KUKA KRL program: EPS_2_25089_SANMH01A_C_20251118074754.src

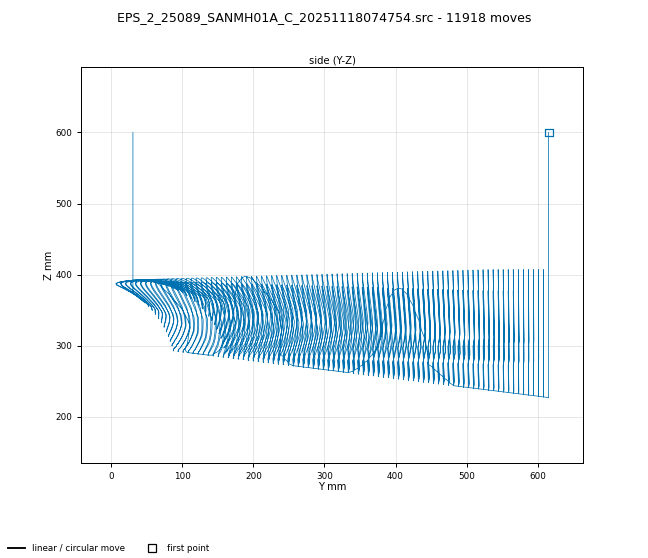
[picture p0: tool path of EPS_2_25089_SANMH01A_C_20251118074754.src, 11918 of 11920 moves have a stored position in this frame; points joined in program order, loops and branches not executed]
&ACCESS RVP
&REL 4
&COMMENT QRS 19112012
&PARAM EDITMASK = *
DEF PART()
EXT BAS (BAS_COMMAND :IN,REAL :IN )
INT I
BAS (#INITMOV,0 )

;KUKA QRS Post kuka4.cps  Date:22-06-2017 !

File_ID=2924

QRS_PRE_INIT()

;Init var - Until changes are made in qrs_pre_init
Outlet_Square_prg=0
Inlet_1_Square_prg=0
Inlet_2_Square_prg=0
Inlet_3_Square_prg=0
Inlet_4_Square_prg=0
Inlet_5_Square_prg=0

Outlet_1={X 0.000, Y 531.880, Z 306.500, B 0.000, E1 0.000 }
Inlet_1={X 0.000, Y 534.050, Z 276.500, B 0.000, E1 193.000 }
Outlet_1_type=201
Inlet_1_type=201
;QRS#1=Sidecore dimensions
;QRS#2=200-8" PVC SDR 35
;QRS#3=200-8" PVC SDR 35
;QRS#4=
;QRS#5=
;QRS#6=
;QRS#7=
;QRS#8=
;QRS#9=12-08 PSX
;QRS#10=12-08 PSX
;QRS#11=
;QRS#12=
;QRS#13=
;QRS#14=
;QRS#15=
;QRS#16=1220x127x686 2,25'
;QRS#17=EPS Height
;QRS#18=407
;QRS#19=*
;QRS#20= UPDATED VERSION 22-06-2017
;QRS#21=*
Outlet_Square=0100
Inlet_1_Square=0100
Inlet_2_Square=0
Inlet_3_Square=0
Inlet_4_Square=0
Inlet_5_Square=0
Mill_Square=1
Outlet_Square_Prg=204
Inlet_1_Square_prg=204

QRS_INIT()

$ADVANCE=5

; T1
PTP {E1 173.593,E2 173.593}
PTP {X 0,Y 615.507,A -85,B 0,C 180,E1 173.593,E2 173.593,E3 0,E4 0,E5 0,E6 0}
QRS_SPEED_INIT()
LIN {X 0,Y 615.507,Z 600,A -85,B 0,C 180,E1 173.593,E2 173.593,E3 0,E4 0,E5 0,E6 0} C_VEL
LIN {X 0,Y 615.507,Z 236.874,A -85,B 0,C 180,E1 173.593,E2 173.593} C_VEL
LIN {X 0,Y 615.507,Z 228.699,A -85,B 0,C 180,E1 173.593,E2 173.593} C_VEL
LIN {X 0,Y 615.492,Z 226.699,A -85,B 0,C 180,E1 173.407,E2 173.407} C_VEL
LIN {X 0,Y 615.497,Z 226.682,A -85,B 0,C 180,E1 170.802,E2 170.802} C_VEL
LIN {X 0,Y 615.47,Z 226.694,A -85,B 0,C 180,E1 168.14,E2 168.14} C_VEL
LIN {X 0,Y 615.478,Z 226.693,A -85,B 0,C 180,E1 165.452,E2 165.452} C_VEL
LIN {X 0,Y 615.483,Z 226.686,A -85,B 0,C 180,E1 162.73,E2 162.73} C_VEL
LIN {X 0,Y 615.486,Z 226.7,A -85,B 0,C 180,E1 159.968,E2 159.968} C_VEL
LIN {X 0,Y 615.487,Z 226.684,A -85,B 0,C 180,E1 157.157,E2 157.157} C_VEL
LIN {X 0,Y 615.497,Z 226.7,A -85,B 0,C 180,E1 154.286,E2 154.286} C_VEL
LIN {X 0,Y 615.486,Z 226.684,A -85,B 0,C 180,E1 151.343,E2 151.343} C_VEL
LIN {X 0,Y 615.486,Z 226.692,A -85,B 0,C 180,E1 148.912,E2 148.912} C_VEL
LIN {X 0,Y 615.482,Z 226.698,A -85,B 0,C 180,E1 146.465,E2 146.465} C_VEL
LIN {X 0,Y 615.482,Z 226.685,A -85,B 0,C 180,E1 143.576,E2 143.576} C_VEL
LIN {X 0,Y 615.497,Z 226.699,A -85,B 0,C 180,E1 140.935,E2 140.935} C_VEL
LIN {X 0,Y 615.464,Z 226.694,A -85,B 0,C 180,E1 138.526,E2 138.526} C_VEL
LIN {X 0,Y 615.487,Z 226.685,A -85,B 0,C 180,E1 135.852,E2 135.852} C_VEL
LIN {X 0,Y 615.478,Z 226.699,A -85,B 0,C 180,E1 133.048,E2 133.048} C_VEL
LIN {X 0,Y 615.453,Z 226.693,A -85,B 0,C 180,E1 130.608,E2 130.608} C_VEL
LIN {X 0,Y 615.48,Z 226.689,A -85,B 0,C 180,E1 128.013,E2 128.013} C_VEL
LIN {X 0,Y 615.496,Z 226.699,A -85,B 0,C 180,E1 125.614,E2 125.614} C_VEL
LIN {X 0,Y 615.458,Z 226.697,A -85,B 0,C 180,E1 123.237,E2 123.237} C_VEL
LIN {X 0,Y 615.443,Z 226.694,A -85,B 0,C 180,E1 120.921,E2 120.921} C_VEL
LIN {X 0,Y 615.471,Z 226.691,A -85,B 0,C 180,E1 118.45,E2 118.45} C_VEL
LIN {X 0,Y 615.454,Z 226.698,A -85,B 0,C 180,E1 115.565,E2 115.565} C_VEL
LIN {X 0,Y 615.445,Z 226.698,A -85,B 0,C 180,E1 113.558,E2 113.558} C_VEL
LIN {X 0,Y 615.493,Z 226.694,A -85,B 0,C 180,E1 112.351,E2 112.351} C_VEL
LIN {X 0,Y 615.457,Z 230.7,A -85,B 0,C 180,E1 110.033,E2 110.033} C_VEL
LIN {X 0,Y 615.474,Z 234.384,A -85,B 0,C 180,E1 107.957,E2 107.957} C_VEL
LIN {X 0,Y 615.463,Z 239.321,A -85,B 0,C 180,E1 105.226,E2 105.226} C_VEL
LIN {X 0,Y 615.494,Z 244.376,A -85,B 0,C 180,E1 102.53,E2 102.53} C_VEL
LIN {X 0,Y 615.48,Z 249.482,A -85,B 0,C 180,E1 99.862,E2 99.862} C_VEL
LIN {X 0,Y 615.464,Z 254.653,A -85,B 0,C 180,E1 97.216,E2 97.216} C_VEL
LIN {X 0,Y 615.491,Z 259.883,A -85,B 0,C 180,E1 94.584,E2 94.584} C_VEL
LIN {X 0,Y 615.468,Z 265.156,A -85,B 0,C 180,E1 91.963,E2 91.963} C_VEL
LIN {X 0,Y 615.47,Z 270.494,A -85,B 0,C 180,E1 89.346,E2 89.346} C_VEL
LIN {X 0,Y 615.49,Z 272.087,A -85,B 0,C 180,E1 88.569,E2 88.569} C_VEL
LIN {X 0,Y 615.475,Z 287.993,A -85,B 0,C 180,E1 88.201,E2 88.201} C_VEL
LIN {X 0,Y 615.457,Z 299.97,A -85,B 0,C 180,E1 87.791,E2 87.791} C_VEL
LIN {X 0,Y 615.485,Z 312.305,A -85,B 0,C 180,E1 87.218,E2 87.218} C_VEL
LIN {X 0,Y 615.497,Z 323.338,A -85,B 0,C 180,E1 86.563,E2 86.563} C_VEL
LIN {X 0,Y 615.498,Z 333.348,A -85,B 0,C 180,E1 85.826,E2 85.826} C_VEL
LIN {X 0,Y 615.497,Z 343.183,A -85,B 0,C 180,E1 84.923,E2 84.923} C_VEL
LIN {X 0,Y 615.497,Z 351.875,A -85,B 0,C 180,E1 83.937,E2 83.937} C_VEL
LIN {X 0,Y 615.498,Z 357.916,A -85,B 0,C 180,E1 83.094,E2 83.094} C_VEL
LIN {X 0,Y 615.495,Z 363.597,A -85,B 0,C 180,E1 82.125,E2 82.125} C_VEL
LIN {X 0,Y 615.498,Z 368.188,A -85,B 0,C 180,E1 81.133,E2 81.133} C_VEL
LIN {X 0,Y 615.496,Z 371.686,A -85,B 0,C 180,E1 80.138,E2 80.138} C_VEL
LIN {X 0,Y 615.496,Z 374.268,A -85,B 0,C 180,E1 79.101,E2 79.101} C_VEL
LIN {X 0,Y 615.494,Z 375.727,A -85,B 0,C 180,E1 78.14,E2 78.14} C_VEL
LIN {X 0,Y 615.497,Z 376.266,A -85,B 0,C 180,E1 77.47,E2 77.47} C_VEL
LIN {X 0,Y 615.495,Z 376.357,A -85,B 0,C 180,E1 76.799,E2 76.799} C_VEL
LIN {X 0,Y 615.497,Z 376.002,A -85,B 0,C 180,E1 76.058,E2 76.058} C_VEL
LIN {X 0,Y 615.496,Z 375.351,A -85,B 0,C 180,E1 75.452,E2 75.452} C_VEL
LIN {X 0,Y 615.495,Z 374.193,A -85,B 0,C 180,E1 74.775,E2 74.775} C_VEL
LIN {X 0,Y 615.494,Z 371.016,A -85,B 0,C 180,E1 73.562,E2 73.562} C_VEL
LIN {X 0,Y 615.498,Z 366.514,A -85,B 0,C 180,E1 72.387,E2 72.387} C_VEL
LIN {X 0,Y 615.497,Z 361.234,A -85,B 0,C 180,E1 71.355,E2 71.355} C_VEL
LIN {X 0,Y 615.496,Z 354.453,A -85,B 0,C 180,E1 70.316,E2 70.316} C_VEL
LIN {X 0,Y 615.494,Z 345.883,A -85,B 0,C 180,E1 69.27,E2 69.27} C_VEL
LIN {X 0,Y 615.497,Z 336.964,A -85,B 0,C 180,E1 68.393,E2 68.393} C_VEL
LIN {X 0,Y 615.499,Z 325.956,A -85,B 0,C 180,E1 67.526,E2 67.526} C_VEL
LIN {X 0,Y 615.442,Z 315.935,A -85,B 0,C 180,E1 66.888,E2 66.888} C_VEL
LIN {X 0,Y 615.437,Z 303.663,A -85,B 0,C 180,E1 66.274,E2 66.274} C_VEL
LIN {X 0,Y 615.477,Z 290.8,A -85,B 0,C 180,E1 65.795,E2 65.795} C_VEL
LIN {X 0,Y 615.485,Z 277.91,A -85,B 0,C 180,E1 65.459,E2 65.459} C_VEL
LIN {X 0,Y 615.477,Z 272.101,A -85,B 0,C 180,E1 65.346,E2 65.346} C_VEL
LIN {X 0,Y 615.431,Z 266.947,A -85,B 0,C 180,E1 62.821,E2 62.821} C_VEL
LIN {X 0,Y 615.43,Z 262.428,A -85,B 0,C 180,E1 60.591,E2 60.591} C_VEL
LIN {X 0,Y 615.447,Z 257.861,A -85,B 0,C 180,E1 58.313,E2 58.313} C_VEL
LIN {X 0,Y 615.494,Z 253.242,A -85,B 0,C 180,E1 55.979,E2 55.979} C_VEL
LIN {X 0,Y 615.46,Z 248.58,A -85,B 0,C 180,E1 53.574,E2 53.574} C_VEL
LIN {X 0,Y 615.424,Z 243.841,A -85,B 0,C 180,E1 51.092,E2 51.092} C_VEL
LIN {X 0,Y 615.425,Z 239.751,A -85,B 0,C 180,E1 48.91,E2 48.91} C_VEL
LIN {X 0,Y 615.468,Z 235.816,A -85,B 0,C 180,E1 46.755,E2 46.755} C_VEL
LIN {X 0,Y 615.484,Z 230.919,A -85,B 0,C 180,E1 43.998,E2 43.998} C_VEL
LIN {X 0,Y 615.492,Z 227.552,A -85,B 0,C 180,E1 42.082,E2 42.082} C_VEL
LIN {X 0,Y 615.47,Z 226.699,A -85,B 0,C 180,E1 41.474,E2 41.474} C_VEL
LIN {X 0,Y 615.479,Z 226.701,A -85,B 0,C 180,E1 38.904,E2 38.904} C_VEL
LIN {X 0,Y 615.487,Z 226.691,A -85,B 0,C 180,E1 36.423,E2 36.423} C_VEL
LIN {X 0,Y 615.475,Z 226.7,A -85,B 0,C 180,E1 34.021,E2 34.021} C_VEL
LIN {X 0,Y 615.495,Z 226.698,A -85,B 0,C 180,E1 31.089,E2 31.089} C_VEL
LIN {X 0,Y 615.49,Z 226.695,A -85,B 0,C 180,E1 28.453,E2 28.453} C_VEL
LIN {X 0,Y 615.459,Z 226.7,A -85,B 0,C 180,E1 25.566,E2 25.566} C_VEL
LIN {X 0,Y 615.49,Z 226.69,A -85,B 0,C 180,E1 22.843,E2 22.843} C_VEL
LIN {X 0,Y 615.449,Z 226.7,A -85,B 0,C 180,E1 20.033,E2 20.033} C_VEL
LIN {X 0,Y 615.488,Z 226.694,A -85,B 0,C 180,E1 17.269,E2 17.269} C_VEL
LIN {X 0,Y 615.485,Z 226.702,A -85,B 0,C 180,E1 14.548,E2 14.548} C_VEL
LIN {X 0,Y 615.469,Z 226.7,A -85,B 0,C 180,E1 11.86,E2 11.86} C_VEL
LIN {X 0,Y 615.497,Z 226.689,A -85,B 0,C 180,E1 9.198,E2 9.198} C_VEL
LIN {X 0,Y 615.453,Z 226.7,A -85,B 0,C 180,E1 6.556,E2 6.556} C_VEL
LIN {X 0,Y 615.49,Z 226.699,A -85,B 0,C 180,E1 3.928,E2 3.928} C_VEL
LIN {X 0,Y 615.496,Z 226.694,A -85,B 0,C 180,E1 1.308,E2 1.308} C_VEL
LIN {X 0,Y 615.447,Z 226.7,A -85,B 0,C 180,E1 -1.309,E2 -1.309} C_VEL
LIN {X 0,Y 615.479,Z 226.695,A -85,B 0,C 180,E1 -3.929,E2 -3.929} C_VEL
LIN {X 0,Y 615.487,Z 226.701,A -85,B 0,C 180,E1 -6.589,E2 -6.589} C_VEL
LIN {X 0,Y 615.47,Z 226.698,A -85,B 0,C 180,E1 -9.2,E2 -9.2} C_VEL
LIN {X 0,Y 615.478,Z 226.693,A -85,B 0,C 180,E1 -11.862,E2 -11.862} C_VEL
LIN {X 0,Y 615.458,Z 226.699,A -85,B 0,C 180,E1 -14.55,E2 -14.55} C_VEL
LIN {X 0,Y 615.487,Z 226.698,A -85,B 0,C 180,E1 -17.271,E2 -17.271} C_VEL
LIN {X 0,Y 615.493,Z 226.699,A -85,B 0,C 180,E1 -20.033,E2 -20.033} C_VEL
LIN {X 0,Y 615.475,Z 226.698,A -85,B 0,C 180,E1 -22.846,E2 -22.846} C_VEL
LIN {X 0,Y 615.493,Z 226.692,A -85,B 0,C 180,E1 -25.716,E2 -25.716} C_VEL
LIN {X 0,Y 615.456,Z 226.699,A -85,B 0,C 180,E1 -28.66,E2 -28.66} C_VEL
LIN {X 0,Y 615.48,Z 226.695,A -85,B 0,C 180,E1 -31.087,E2 -31.087} C_VEL
LIN {X 0,Y 615.494,Z 226.697,A -85,B 0,C 180,E1 -33.537,E2 -33.537} C_VEL
LIN {X 0,Y 615.475,Z 226.698,A -85,B 0,C 180,E1 -36.426,E2 -36.426} C_VEL
LIN {X 0,Y 615.473,Z 226.694,A -85,B 0,C 180,E1 -39.062,E2 -39.062} C_VEL
LIN {X 0,Y 615.481,Z 226.698,A -85,B 0,C 180,E1 -41.475,E2 -41.475} C_VEL
LIN {X 0,Y 615.491,Z 226.699,A -85,B 0,C 180,E1 -44.15,E2 -44.15} C_VEL
LIN {X 0,Y 615.472,Z 226.698,A -85,B 0,C 180,E1 -46.955,E2 -46.955} C_VEL
LIN {X 0,Y 615.473,Z 226.695,A -85,B 0,C 180,E1 -49.394,E2 -49.394} C_VEL
LIN {X 0,Y 615.483,Z 226.699,A -85,B 0,C 180,E1 -51.989,E2 -51.989} C_VEL
LIN {X 0,Y 615.471,Z 226.817,A -85,B 0,C 180,E1 -54.585,E2 -54.585} C_VEL
LIN {X 0,Y 615.487,Z 233.979,A -85,B 0,C 180,E1 -57.155,E2 -57.155} C_VEL
LIN {X 0,Y 615.451,Z 241.781,A -85,B 0,C 180,E1 -59.839,E2 -59.839} C_VEL
LIN {X 0,Y 615.493,Z 249.545,A -85,B 0,C 180,E1 -62.455,E2 -62.455} C_VEL
LIN {X 0,Y 615.47,Z 257.31,A -85,B 0,C 180,E1 -65.008,E2 -65.008} C_VEL
LIN {X 0,Y 615.475,Z 265.53,A -85,B 0,C 180,E1 -67.658,E2 -67.658} C_VEL
LIN {X 0,Y 615.486,Z 273.928,A -85,B 0,C 180,E1 -70.316,E2 -70.316} C_VEL
LIN {X 0,Y 615.488,Z 282.785,A -85,B 0,C 180,E1 -73.072,E2 -73.072} C_VEL
LIN {X 0,Y 615.46,Z 291.558,A -85,B 0,C 180,E1 -75.763,E2 -75.763} C_VEL
LIN {X 0,Y 615.498,Z 300.138,A -85,B 0,C 180,E1 -78.369,E2 -78.369} C_VEL
LIN {X 0,Y 615.497,Z 313.833,A -85,B 0,C 180,E1 -78.641,E2 -78.641} C_VEL
LIN {X 0,Y 615.451,Z 327.002,A -85,B 0,C 180,E1 -79.052,E2 -79.052} C_VEL
LIN {X 0,Y 615.438,Z 338.78,A -85,B 0,C 180,E1 -79.556,E2 -79.556} C_VEL
LIN {X 0,Y 615.482,Z 349.393,A -85,B 0,C 180,E1 -80.138,E2 -80.138} C_VEL
LIN {X 0,Y 615.498,Z 360.235,A -85,B 0,C 180,E1 -80.884,E2 -80.884} C_VEL
LIN {X 0,Y 615.497,Z 370.814,A -85,B 0,C 180,E1 -81.794,E2 -81.794} C_VEL
LIN {X 0,Y 615.498,Z 378.608,A -85,B 0,C 180,E1 -82.62,E2 -82.62} C_VEL
LIN {X 0,Y 615.496,Z 386.204,A -85,B 0,C 180,E1 -83.608,E2 -83.608} C_VEL
LIN {X 0,Y 615.498,Z 393.205,A -85,B 0,C 180,E1 -84.759,E2 -84.759} C_VEL
LIN {X 0,Y 615.494,Z 397.852,A -85,B 0,C 180,E1 -85.744,E2 -85.744} C_VEL
LIN {X 0,Y 615.494,Z 401.399,A -85,B 0,C 180,E1 -86.727,E2 -86.727} C_VEL
LIN {X 0,Y 615.497,Z 403.233,A -85,B 0,C 180,E1 -87.382,E2 -87.382} C_VEL
LIN {X 0,Y 615.5,Z 404.608,A -85,B 0,C 180,E1 -88.037,E2 -88.037} C_VEL
LIN {X 0,Y 615.496,Z 406.174,A -85,B 0,C 180,E1 -89.346,E2 -89.346} C_VEL
LIN {X 0,Y 615.494,Z 406.389,A -85,B 0,C 180,E1 -90,E2 -90} C_VEL
LIN {X 0,Y 615.495,Z 405.58,A -85,B 0,C 180,E1 -91.309,E2 -91.309} C_VEL
LIN {X 0,Y 615.5,Z 404.607,A -85,B 0,C 180,E1 -91.963,E2 -91.963} C_VEL
LIN {X 0,Y 615.497,Z 403.233,A -85,B 0,C 180,E1 -92.618,E2 -92.618} C_VEL
LIN {X 0,Y 615.496,Z 400.35,A -85,B 0,C 180,E1 -93.601,E2 -93.601} C_VEL
LIN {X 0,Y 615.498,Z 396.442,A -85,B 0,C 180,E1 -94.584,E2 -94.584} C_VEL
LIN {X 0,Y 615.499,Z 391.405,A -85,B 0,C 180,E1 -95.57,E2 -95.57} C_VEL
LIN {X 0,Y 615.497,Z 384.871,A -85,B 0,C 180,E1 -96.583,E2 -96.583} C_VEL
LIN {X 0,Y 615.497,Z 377.134,A -85,B 0,C 180,E1 -97.545,E2 -97.545} C_VEL
LIN {X 0,Y 615.498,Z 369.047,A -85,B 0,C 180,E1 -98.371,E2 -98.371} C_VEL
LIN {X 0,Y 615.499,Z 359.17,A -85,B 0,C 180,E1 -99.198,E2 -99.198} C_VEL
LIN {X 0,Y 615.472,Z 347.988,A -85,B 0,C 180,E1 -99.945,E2 -99.945} C_VEL
LIN {X 0,Y 615.437,Z 337.035,A -85,B 0,C 180,E1 -100.528,E2 -100.528} C_VEL
LIN {X 0,Y 615.457,Z 324.799,A -85,B 0,C 180,E1 -101.03,E2 -101.03} C_VEL
LIN {X 0,Y 615.499,Z 312.073,A -85,B 0,C 180,E1 -101.401,E2 -101.401} C_VEL
LIN {X 0,Y 615.498,Z 300.138,A -85,B 0,C 180,E1 -101.631,E2 -101.631} C_VEL
LIN {X 0,Y 615.46,Z 291.558,A -85,B 0,C 180,E1 -104.237,E2 -104.237} C_VEL
LIN {X 0,Y 615.488,Z 282.785,A -85,B 0,C 180,E1 -106.928,E2 -106.928} C_VEL
LIN {X 0,Y 615.486,Z 273.928,A -85,B 0,C 180,E1 -109.685,E2 -109.685} C_VEL
LIN {X 0,Y 615.479,Z 265.527,A -85,B 0,C 180,E1 -112.343,E2 -112.343} C_VEL
LIN {X 0,Y 615.47,Z 257.31,A -85,B 0,C 180,E1 -114.992,E2 -114.992} C_VEL
LIN {X 0,Y 615.453,Z 248.442,A -85,B 0,C 180,E1 -117.916,E2 -117.916} C_VEL
LIN {X 0,Y 615.473,Z 240.661,A -85,B 0,C 180,E1 -120.539,E2 -120.539} C_VEL
LIN {X 0,Y 615.491,Z 232.875,A -85,B 0,C 180,E1 -123.235,E2 -123.235} C_VEL
LIN {X 0,Y 615.453,Z 226.699,A -85,B 0,C 180,E1 -125.517,E2 -125.517} C_VEL
LIN {X 0,Y 615.419,Z 226.699,A -85,B 0,C 180,E1 -128.003,E2 -128.003} C_VEL
LIN {X 0,Y 615.421,Z 226.699,A -85,B 0,C 180,E1 -130.081,E2 -130.081} C_VEL
LIN {X 0,Y 615.439,Z 226.699,A -85,B 0,C 180,E1 -132.356,E2 -132.356} C_VEL
LIN {X 0,Y 615.454,Z 226.7,A -85,B 0,C 180,E1 -135.07,E2 -135.07} C_VEL
LIN {X 0,Y 615.462,Z 226.699,A -85,B 0,C 180,E1 -136.954,E2 -136.954} C_VEL
LIN {X 0,Y 615.423,Z 226.699,A -85,B 0,C 180,E1 -139.388,E2 -139.388} C_VEL
LIN {X 0,Y 615.444,Z 226.699,A -85,B 0,C 180,E1 -141.992,E2 -141.992} C_VEL
LIN {X 0,Y 615.5,Z 226.699,A -85,B 0,C 180,E1 -144.384,E2 -144.384} C_VEL
LIN {X 0,Y 615.457,Z 226.695,A -85,B 0,C 180,E1 -146.761,E2 -146.761} C_VEL
LIN {X 0,Y 615.434,Z 226.696,A -85,B 0,C 180,E1 -149.077,E2 -149.077} C_VEL
LIN {X 0,Y 615.448,Z 226.698,A -85,B 0,C 180,E1 -151.554,E2 -151.554} C_VEL
LIN {X 0,Y 615.472,Z 226.691,A -85,B 0,C 180,E1 -154.432,E2 -154.432} C_VEL
LIN {X 0,Y 615.466,Z 226.691,A -85,B 0,C 180,E1 -156.442,E2 -156.442} C_VEL
LIN {X 0,Y 615.453,Z 226.692,A -85,B 0,C 180,E1 -158.566,E2 -158.566} C_VEL
LIN {X 0,Y 615.447,Z 226.693,A -85,B 0,C 180,E1 -160.66,E2 -160.66} C_VEL
LIN {X 0,Y 615.447,Z 226.693,A -85,B 0,C 180,E1 -162.728,E2 -162.728} C_VEL
LIN {X 0,Y 615.489,Z 226.702,A -85,B 0,C 180,E1 -165.45,E2 -165.45} C_VEL
LIN {X 0,Y 615.469,Z 226.688,A -85,B 0,C 180,E1 -168.138,E2 -168.138} C_VEL
LIN {X 0,Y 615.464,Z 226.696,A -85,B 0,C 180,E1 -170.8,E2 -170.8} C_VEL
LIN {X 0,Y 615.493,Z 226.69,A -85,B 0,C 180,E1 -173.443,E2 -173.443} C_VEL
LIN {X 0,Y 615.464,Z 226.689,A -85,B 0,C 180,E1 -176.071,E2 -176.071} C_VEL
LIN {X 0,Y 615.481,Z 226.699,A -85,B 0,C 180,E1 -178.691,E2 -178.691} C_VEL
LIN {X 0,Y 615.492,Z 226.686,A -85,B 0,C 180,E1 -181.308,E2 -181.308} C_VEL
LIN {X 0,Y 615.467,Z 226.69,A -85,B 0,C 180,E1 -183.928,E2 -183.928} C_VEL
LIN {X 0,Y 615.492,Z 226.699,A -85,B 0,C 180,E1 -186.593,E2 -186.593} C_VEL
LIN {X 0,Y 614.815,Z 226.834,A -85,B 0,C 180,E1 -187.139,E2 -187.139} C_VEL
LIN {X 0,Y 611.985,Z 227.251,A -85,B 0,C 180,E1 -188.025,E2 -188.025} C_VEL
LIN {X 0,Y 609.593,Z 227.559,A -85,B 0,C 180,E1 -188.737,E2 -188.737} C_VEL
LIN {X 0,Y 608.552,Z 227.677,A -85,B 0,C 180,E1 -189.287,E2 -189.287} C_VEL
LIN {X 0,Y 608.459,Z 227.687,A -85,B 0,C 180,E1 -189.473,E2 -189.473} C_VEL
LIN {X 0,Y 608.449,Z 227.694,A -85,B 0,C 180,E1 -191.999,E2 -191.999} C_VEL
LIN {X 0,Y 608.468,Z 227.688,A -85,B 0,C 180,E1 -194.72,E2 -194.72} C_VEL
LIN {X 0,Y 608.45,Z 227.69,A -85,B 0,C 180,E1 -197.476,E2 -197.476} C_VEL
LIN {X 0,Y 608.459,Z 227.692,A -85,B 0,C 180,E1 -200.273,E2 -200.273} C_VEL
LIN {X 0,Y 608.45,Z 227.689,A -85,B 0,C 180,E1 -203.123,E2 -203.123} C_VEL
LIN {X 0,Y 608.474,Z 227.695,A -85,B 0,C 180,E1 -205.724,E2 -205.724} C_VEL
LIN {X 0,Y 608.467,Z 227.686,A -85,B 0,C 180,E1 -208.621,E2 -208.621} C_VEL
LIN {X 0,Y 608.467,Z 227.694,A -85,B 0,C 180,E1 -211.315,E2 -211.315} C_VEL
LIN {X 0,Y 608.463,Z 227.691,A -85,B 0,C 180,E1 -213.735,E2 -213.735} C_VEL
LIN {X 0,Y 608.463,Z 227.687,A -85,B 0,C 180,E1 -216.09,E2 -216.09} C_VEL
LIN {X 0,Y 608.465,Z 227.689,A -85,B 0,C 180,E1 -218.587,E2 -218.587} C_VEL
LIN {X 0,Y 608.45,Z 227.693,A -85,B 0,C 180,E1 -221.342,E2 -221.342} C_VEL
LIN {X 0,Y 608.457,Z 227.687,A -85,B 0,C 180,E1 -223.869,E2 -223.869} C_VEL
LIN {X 0,Y 608.483,Z 227.693,A -85,B 0,C 180,E1 -226.688,E2 -226.688} C_VEL
LIN {X 0,Y 608.437,Z 227.69,A -85,B 0,C 180,E1 -229.697,E2 -229.697} C_VEL
LIN {X 0,Y 608.461,Z 227.692,A -85,B 0,C 180,E1 -232.254,E2 -232.254} C_VEL
LIN {X 0,Y 608.433,Z 227.696,A -85,B 0,C 180,E1 -234.723,E2 -234.723} C_VEL
LIN {X 0,Y 608.433,Z 227.691,A -85,B 0,C 180,E1 -237.12,E2 -237.12} C_VEL
LIN {X 0,Y 608.481,Z 227.695,A -85,B 0,C 180,E1 -240.222,E2 -240.222} C_VEL
LIN {X 0,Y 608.417,Z 227.693,A -85,B 0,C 180,E1 -242.801,E2 -242.801} C_VEL
LIN {X 0,Y 608.437,Z 227.692,A -85,B 0,C 180,E1 -245.429,E2 -245.429} C_VEL
LIN {X 0,Y 608.463,Z 227.692,A -85,B 0,C 180,E1 -247.595,E2 -247.595} C_VEL
LIN {X 0,Y 608.449,Z 231.225,A -85,B 0,C 180,E1 -249.726,E2 -249.726} C_VEL
LIN {X 0,Y 608.441,Z 234.929,A -85,B 0,C 180,E1 -251.828,E2 -251.828} C_VEL
LIN {X 0,Y 608.445,Z 238.634,A -85,B 0,C 180,E1 -253.906,E2 -253.906} C_VEL
LIN {X 0,Y 608.413,Z 243.672,A -85,B 0,C 180,E1 -256.643,E2 -256.643} C_VEL
LIN {X 0,Y 608.432,Z 248.794,A -85,B 0,C 180,E1 -259.35,E2 -259.35} C_VEL
LIN {X 0,Y 608.437,Z 253.977,A -85,B 0,C 180,E1 -262.033,E2 -262.033} C_VEL
LIN {X 0,Y 608.43,Z 259.22,A -85,B 0,C 180,E1 -264.698,E2 -264.698} C_VEL
LIN {X 0,Y 608.425,Z 264.522,A -85,B 0,C 180,E1 -267.352,E2 -267.352} C_VEL
LIN {X 0,Y 608.407,Z 269.882,A -85,B 0,C 180,E1 -270,E2 -270} C_VEL
LIN {X 0,Y 608.427,Z 272.54,A -85,B 0,C 180,E1 -271.303,E2 -271.303} C_VEL
LIN {X 0,Y 608.523,Z 287.576,A -85,B 0,C 180,E1 -271.654,E2 -271.654} C_VEL
LIN {X 0,Y 608.478,Z 299.736,A -85,B 0,C 180,E1 -272.068,E2 -272.068} C_VEL
LIN {X 0,Y 608.493,Z 310.656,A -85,B 0,C 180,E1 -272.565,E2 -272.565} C_VEL
LIN {X 0,Y 608.486,Z 322.069,A -85,B 0,C 180,E1 -273.228,E2 -273.228} C_VEL
LIN {X 0,Y 608.472,Z 332.38,A -85,B 0,C 180,E1 -273.974,E2 -273.974} C_VEL
LIN {X 0,Y 608.463,Z 341.737,A -85,B 0,C 180,E1 -274.803,E2 -274.803} C_VEL
LIN {X 0,Y 608.458,Z 350.779,A -85,B 0,C 180,E1 -275.8,E2 -275.8} C_VEL
LIN {X 0,Y 608.453,Z 358.102,A -85,B 0,C 180,E1 -276.799,E2 -276.799} C_VEL
LIN {X 0,Y 608.447,Z 363.081,A -85,B 0,C 180,E1 -277.633,E2 -277.633} C_VEL
LIN {X 0,Y 608.428,Z 367.93,A -85,B 0,C 180,E1 -278.636,E2 -278.636} C_VEL
LIN {X 0,Y 608.427,Z 371.661,A -85,B 0,C 180,E1 -279.642,E2 -279.642} C_VEL
LIN {X 0,Y 608.451,Z 375.02,A -85,B 0,C 180,E1 -280.954,E2 -280.954} C_VEL
LIN {X 0,Y 608.437,Z 376.507,A -85,B 0,C 180,E1 -282,E2 -282} C_VEL
LIN {X 0,Y 608.418,Z 376.92,A -85,B 0,C 180,E1 -282.678,E2 -282.678} C_VEL
LIN {X 0,Y 608.43,Z 376.572,A -85,B 0,C 180,E1 -284.008,E2 -284.008} C_VEL
LIN {X 0,Y 608.419,Z 375.715,A -85,B 0,C 180,E1 -284.722,E2 -284.722} C_VEL
LIN {X 0,Y 608.419,Z 374.443,A -85,B 0,C 180,E1 -285.407,E2 -285.407} C_VEL
LIN {X 0,Y 608.425,Z 371.433,A -85,B 0,C 180,E1 -286.52,E2 -286.52} C_VEL
LIN {X 0,Y 608.428,Z 367.832,A -85,B 0,C 180,E1 -287.477,E2 -287.477} C_VEL
LIN {X 0,Y 608.444,Z 363.155,A -85,B 0,C 180,E1 -288.443,E2 -288.443} C_VEL
LIN {X 0,Y 608.469,Z 356.225,A -85,B 0,C 180,E1 -289.569,E2 -289.569} C_VEL
LIN {X 0,Y 608.459,Z 348.688,A -85,B 0,C 180,E1 -290.542,E2 -290.542} C_VEL
LIN {X 0,Y 608.466,Z 339.341,A -85,B 0,C 180,E1 -291.513,E2 -291.513} C_VEL
LIN {X 0,Y 608.49,Z 329.866,A -85,B 0,C 180,E1 -292.315,E2 -292.315} C_VEL
LIN {X 0,Y 608.459,Z 319.398,A -85,B 0,C 180,E1 -293.033,E2 -293.033} C_VEL
LIN {X 0,Y 608.444,Z 307.812,A -85,B 0,C 180,E1 -293.664,E2 -293.664} C_VEL
LIN {X 0,Y 608.513,Z 295.153,A -85,B 0,C 180,E1 -294.193,E2 -294.193} C_VEL
LIN {X 0,Y 608.537,Z 282.691,A -85,B 0,C 180,E1 -294.567,E2 -294.567} C_VEL
LIN {X 0,Y 608.411,Z 272.608,A -85,B 0,C 180,E1 -294.777,E2 -294.777} C_VEL
LIN {X 0,Y 608.387,Z 266.981,A -85,B 0,C 180,E1 -297.52,E2 -297.52} C_VEL
LIN {X 0,Y 608.433,Z 262.055,A -85,B 0,C 180,E1 -299.968,E2 -299.968} C_VEL
LIN {X 0,Y 608.39,Z 256.28,A -85,B 0,C 180,E1 -302.883,E2 -302.883} C_VEL
LIN {X 0,Y 608.376,Z 251.604,A -85,B 0,C 180,E1 -305.281,E2 -305.281} C_VEL
LIN {X 0,Y 608.398,Z 246.871,A -85,B 0,C 180,E1 -307.75,E2 -307.75} C_VEL
LIN {X 0,Y 608.416,Z 242.032,A -85,B 0,C 180,E1 -310.327,E2 -310.327} C_VEL
LIN {X 0,Y 608.417,Z 237.242,A -85,B 0,C 180,E1 -312.962,E2 -312.962} C_VEL
LIN {X 0,Y 608.459,Z 232.33,A -85,B 0,C 180,E1 -315.735,E2 -315.735} C_VEL
LIN {X 0,Y 608.468,Z 228.482,A -85,B 0,C 180,E1 -317.941,E2 -317.941} C_VEL
LIN {X 0,Y 608.427,Z 227.696,A -85,B 0,C 180,E1 -318.823,E2 -318.823} C_VEL
LIN {X 0,Y 608.454,Z 227.692,A -85,B 0,C 180,E1 -321.76,E2 -321.76} C_VEL
LIN {X 0,Y 608.469,Z 227.692,A -85,B 0,C 180,E1 -323.95,E2 -323.95} C_VEL
LIN {X 0,Y 608.426,Z 227.696,A -85,B 0,C 180,E1 -326.328,E2 -326.328} C_VEL
LIN {X 0,Y 608.468,Z 227.695,A -85,B 0,C 180,E1 -328.727,E2 -328.727} C_VEL
LIN {X 0,Y 608.475,Z 227.69,A -85,B 0,C 180,E1 -331.377,E2 -331.377} C_VEL
LIN {X 0,Y 608.443,Z 227.694,A -85,B 0,C 180,E1 -334.282,E2 -334.282} C_VEL
LIN {X 0,Y 608.452,Z 227.693,A -85,B 0,C 180,E1 -336.877,E2 -336.877} C_VEL
LIN {X 0,Y 608.442,Z 227.695,A -85,B 0,C 180,E1 -339.726,E2 -339.726} C_VEL
LIN {X 0,Y 608.447,Z 227.697,A -85,B 0,C 180,E1 -342.524,E2 -342.524} C_VEL
LIN {X 0,Y 608.472,Z 227.694,A -85,B 0,C 180,E1 -345.28,E2 -345.28} C_VEL
LIN {X 0,Y 608.441,Z 227.695,A -85,B 0,C 180,E1 -348.001,E2 -348.001} C_VEL
LIN {X 0,Y 608.478,Z 227.689,A -85,B 0,C 180,E1 -350.695,E2 -350.695} C_VEL
LIN {X 0,Y 608.425,Z 227.696,A -85,B 0,C 180,E1 -353.4,E2 -353.4} C_VEL
LIN {X 0,Y 608.457,Z 227.697,A -85,B 0,C 180,E1 -356.027,E2 -356.027} C_VEL
LIN {X 0,Y 608.477,Z 227.691,A -85,B 0,C 180,E1 -358.677,E2 -358.677} C_VEL
LIN {X 0,Y 608.435,Z 227.694,A -85,B 0,C 180,E1 -361.325,E2 -361.325} C_VEL
LIN {X 0,Y 608.449,Z 227.693,A -85,B 0,C 180,E1 -363.975,E2 -363.975} C_VEL
LIN {X 0,Y 608.466,Z 227.695,A -85,B 0,C 180,E1 -366.633,E2 -366.633} C_VEL
LIN {X 0,Y 608.457,Z 227.694,A -85,B 0,C 180,E1 -369.307,E2 -369.307} C_VEL
LIN {X 0,Y 608.456,Z 227.692,A -85,B 0,C 180,E1 -372.001,E2 -372.001} C_VEL
LIN {X 0,Y 608.422,Z 227.696,A -85,B 0,C 180,E1 -374.722,E2 -374.722} C_VEL
LIN {X 0,Y 608.454,Z 227.693,A -85,B 0,C 180,E1 -377.477,E2 -377.477} C_VEL
LIN {X 0,Y 608.452,Z 227.696,A -85,B 0,C 180,E1 -380.275,E2 -380.275} C_VEL
LIN {X 0,Y 608.445,Z 227.699,A -85,B 0,C 180,E1 -383.125,E2 -383.125} C_VEL
LIN {X 0,Y 608.472,Z 227.691,A -85,B 0,C 180,E1 -385.724,E2 -385.724} C_VEL
LIN {X 0,Y 608.445,Z 227.693,A -85,B 0,C 180,E1 -388.618,E2 -388.618} C_VEL
LIN {X 0,Y 608.472,Z 227.69,A -85,B 0,C 180,E1 -391.317,E2 -391.317} C_VEL
LIN {X 0,Y 608.47,Z 227.696,A -85,B 0,C 180,E1 -393.737,E2 -393.737} C_VEL
LIN {X 0,Y 608.439,Z 227.694,A -85,B 0,C 180,E1 -396.093,E2 -396.093} C_VEL
LIN {X 0,Y 608.46,Z 227.693,A -85,B 0,C 180,E1 -398.589,E2 -398.589} C_VEL
LIN {X 0,Y 608.455,Z 227.697,A -85,B 0,C 180,E1 -401.343,E2 -401.343} C_VEL
LIN {X 0,Y 608.459,Z 227.697,A -85,B 0,C 180,E1 -404.266,E2 -404.266} C_VEL
LIN {X 0,Y 608.437,Z 227.697,A -85,B 0,C 180,E1 -407.04,E2 -407.04} C_VEL
LIN {X 0,Y 608.45,Z 227.693,A -85,B 0,C 180,E1 -409.698,E2 -409.698} C_VEL
LIN {X 0,Y 608.465,Z 227.692,A -85,B 0,C 180,E1 -412.255,E2 -412.255} C_VEL
LIN {X 0,Y 608.448,Z 227.803,A -85,B 0,C 180,E1 -414.47,E2 -414.47} C_VEL
LIN {X 0,Y 608.495,Z 235.11,A -85,B 0,C 180,E1 -417.124,E2 -417.124} C_VEL
LIN {X 0,Y 608.472,Z 241.814,A -85,B 0,C 180,E1 -419.456,E2 -419.456} C_VEL
LIN {X 0,Y 608.441,Z 249.641,A -85,B 0,C 180,E1 -422.109,E2 -422.109} C_VEL
LIN {X 0,Y 608.455,Z 258.545,A -85,B 0,C 180,E1 -425.065,E2 -425.065} C_VEL
LIN {X 0,Y 608.439,Z 266.337,A -85,B 0,C 180,E1 -427.594,E2 -427.594} C_VEL
LIN {X 0,Y 608.46,Z 275.241,A -85,B 0,C 180,E1 -430.43,E2 -430.43} C_VEL
LIN {X 0,Y 608.452,Z 284.145,A -85,B 0,C 180,E1 -433.216,E2 -433.216} C_VEL
LIN {X 0,Y 608.438,Z 293.16,A -85,B 0,C 180,E1 -435.996,E2 -435.996} C_VEL
LIN {X 0,Y 608.436,Z 300.493,A -85,B 0,C 180,E1 -438.233,E2 -438.233} C_VEL
LIN {X 0,Y 608.558,Z 313.945,A -85,B 0,C 180,E1 -438.509,E2 -438.509} C_VEL
LIN {X 0,Y 608.487,Z 325.999,A -85,B 0,C 180,E1 -438.883,E2 -438.883} C_VEL
LIN {X 0,Y 608.467,Z 338.927,A -85,B 0,C 180,E1 -439.435,E2 -439.435} C_VEL
LIN {X 0,Y 608.471,Z 349.583,A -85,B 0,C 180,E1 -440.023,E2 -440.023} C_VEL
LIN {X 0,Y 608.483,Z 360.477,A -85,B 0,C 180,E1 -440.778,E2 -440.778} C_VEL
LIN {X 0,Y 608.475,Z 371.114,A -85,B 0,C 180,E1 -441.699,E2 -441.699} C_VEL
LIN {X 0,Y 608.471,Z 378.962,A -85,B 0,C 180,E1 -442.534,E2 -442.534} C_VEL
LIN {X 0,Y 608.461,Z 386.288,A -85,B 0,C 180,E1 -443.485,E2 -443.485} C_VEL
LIN {X 0,Y 608.451,Z 391.867,A -85,B 0,C 180,E1 -444.366,E2 -444.366} C_VEL
LIN {X 0,Y 608.432,Z 396.951,A -85,B 0,C 180,E1 -445.362,E2 -445.362} C_VEL
LIN {X 0,Y 608.449,Z 400.897,A -85,B 0,C 180,E1 -446.358,E2 -446.358} C_VEL
LIN {X 0,Y 608.425,Z 403.809,A -85,B 0,C 180,E1 -447.352,E2 -447.352} C_VEL
LIN {X 0,Y 608.444,Z 405.201,A -85,B 0,C 180,E1 -448.014,E2 -448.014} C_VEL
LIN {X 0,Y 608.438,Z 406.783,A -85,B 0,C 180,E1 -449.338,E2 -449.338} C_VEL
LIN {X 0,Y 608.434,Z 407,A -85,B 0,C 180,E1 -450,E2 -450} C_VEL
LIN {X 0,Y 608.448,Z 406.184,A -85,B 0,C 180,E1 -451.324,E2 -451.324} C_VEL
LIN {X 0,Y 608.445,Z 405.201,A -85,B 0,C 180,E1 -451.986,E2 -451.986} C_VEL
LIN {X 0,Y 608.425,Z 403.809,A -85,B 0,C 180,E1 -452.648,E2 -452.648} C_VEL
LIN {X 0,Y 608.449,Z 400.896,A -85,B 0,C 180,E1 -453.642,E2 -453.642} C_VEL
LIN {X 0,Y 608.432,Z 396.95,A -85,B 0,C 180,E1 -454.638,E2 -454.638} C_VEL
LIN {X 0,Y 608.438,Z 390.877,A -85,B 0,C 180,E1 -455.801,E2 -455.801} C_VEL
LIN {X 0,Y 608.462,Z 384.236,A -85,B 0,C 180,E1 -456.799,E2 -456.799} C_VEL
LIN {X 0,Y 608.456,Z 375.99,A -85,B 0,C 180,E1 -457.8,E2 -457.8} C_VEL
LIN {X 0,Y 608.472,Z 367.538,A -85,B 0,C 180,E1 -458.636,E2 -458.636} C_VEL
LIN {X 0,Y 608.48,Z 357.093,A -85,B 0,C 180,E1 -459.473,E2 -459.473} C_VEL
LIN {X 0,Y 608.482,Z 346.759,A -85,B 0,C 180,E1 -460.145,E2 -460.145} C_VEL
LIN {X 0,Y 608.463,Z 335.876,A -85,B 0,C 180,E1 -460.712,E2 -460.712} C_VEL
LIN {X 0,Y 608.492,Z 324.106,A -85,B 0,C 180,E1 -461.186,E2 -461.186} C_VEL
LIN {X 0,Y 608.551,Z 311.277,A -85,B 0,C 180,E1 -461.554,E2 -461.554} C_VEL
LIN {X 0,Y 608.436,Z 300.493,A -85,B 0,C 180,E1 -461.768,E2 -461.768} C_VEL
LIN {X 0,Y 608.407,Z 291.936,A -85,B 0,C 180,E1 -464.38,E2 -464.38} C_VEL
LIN {X 0,Y 608.452,Z 284.145,A -85,B 0,C 180,E1 -466.784,E2 -466.784} C_VEL
LIN {X 0,Y 608.459,Z 275.241,A -85,B 0,C 180,E1 -469.57,E2 -469.57} C_VEL
LIN {X 0,Y 608.461,Z 266.117,A -85,B 0,C 180,E1 -472.476,E2 -472.476} C_VEL
LIN {X 0,Y 608.451,Z 257.432,A -85,B 0,C 180,E1 -475.3,E2 -475.3} C_VEL
LIN {X 0,Y 608.441,Z 249.641,A -85,B 0,C 180,E1 -477.891,E2 -477.891} C_VEL
LIN {X 0,Y 608.472,Z 241.811,A -85,B 0,C 180,E1 -480.544,E2 -480.544} C_VEL
LIN {X 0,Y 608.52,Z 234.014,A -85,B 0,C 180,E1 -483.27,E2 -483.27} C_VEL
LIN {X 0,Y 608.425,Z 227.696,A -85,B 0,C 180,E1 -485.583,E2 -485.583} C_VEL
LIN {X 0,Y 608.425,Z 227.693,A -85,B 0,C 180,E1 -487.748,E2 -487.748} C_VEL
LIN {X 0,Y 608.43,Z 227.692,A -85,B 0,C 180,E1 -490.326,E2 -490.326} C_VEL
LIN {X 0,Y 608.434,Z 227.693,A -85,B 0,C 180,E1 -493.305,E2 -493.305} C_VEL
LIN {X 0,Y 608.421,Z 227.694,A -85,B 0,C 180,E1 -496.126,E2 -496.126} C_VEL
LIN {X 0,Y 608.437,Z 227.696,A -85,B 0,C 180,E1 -498.821,E2 -498.821} C_VEL
LIN {X 0,Y 608.4,Z 227.696,A -85,B 0,C 180,E1 -501.766,E2 -501.766} C_VEL
LIN {X 0,Y 608.432,Z 227.694,A -85,B 0,C 180,E1 -503.955,E2 -503.955} C_VEL
LIN {X 0,Y 608.459,Z 227.696,A -85,B 0,C 180,E1 -506.328,E2 -506.328} C_VEL
LIN {X 0,Y 608.43,Z 227.693,A -85,B 0,C 180,E1 -508.733,E2 -508.733} C_VEL
LIN {X 0,Y 608.409,Z 227.693,A -85,B 0,C 180,E1 -510.976,E2 -510.976} C_VEL
LIN {X 0,Y 608.405,Z 227.695,A -85,B 0,C 180,E1 -513.223,E2 -513.223} C_VEL
LIN {X 0,Y 608.48,Z 227.695,A -85,B 0,C 180,E1 -515.844,E2 -515.844} C_VEL
LIN {X 0,Y 608.452,Z 227.69,A -85,B 0,C 180,E1 -518.307,E2 -518.307} C_VEL
LIN {X 0,Y 608.438,Z 227.693,A -85,B 0,C 180,E1 -521.129,E2 -521.129} C_VEL
LIN {X 0,Y 608.459,Z 227.691,A -85,B 0,C 180,E1 -523.905,E2 -523.905} C_VEL
LIN {X 0,Y 608.436,Z 227.691,A -85,B 0,C 180,E1 -526.642,E2 -526.642} C_VEL
LIN {X 0,Y 608.467,Z 227.695,A -85,B 0,C 180,E1 -529.35,E2 -529.35} C_VEL
LIN {X 0,Y 608.461,Z 227.687,A -85,B 0,C 180,E1 -532.032,E2 -532.032} C_VEL
LIN {X 0,Y 608.452,Z 227.693,A -85,B 0,C 180,E1 -534.697,E2 -534.697} C_VEL
LIN {X 0,Y 608.481,Z 227.688,A -85,B 0,C 180,E1 -537.351,E2 -537.351} C_VEL
LIN {X 0,Y 608.457,Z 227.688,A -85,B 0,C 180,E1 -539.999,E2 -539.999} C_VEL
LIN {X 0,Y 608.477,Z 227.695,A -85,B 0,C 180,E1 -542.647,E2 -542.647} C_VEL
LIN {X 0,Y 608.469,Z 227.687,A -85,B 0,C 180,E1 -545.301,E2 -545.301} C_VEL
LIN {X 0,Y 608.464,Z 227.689,A -85,B 0,C 180,E1 -547.966,E2 -547.966} C_VEL
LIN {X 0,Y 608.459,Z 227.687,A -85,B 0,C 180,E1 -549.473,E2 -549.473} C_VEL
LIN {X 0,Y 607.77,Z 227.779,A -85,B 0,C 180,E1 -550.025,E2 -550.025} C_VEL
LIN {X 0,Y 604.908,Z 228.137,A -85,B 0,C 180,E1 -550.922,E2 -550.922} C_VEL
LIN {X 0,Y 602.507,Z 228.438,A -85,B 0,C 180,E1 -551.644,E2 -551.644} C_VEL
LIN {X 0,Y 601.483,Z 228.565,A -85,B 0,C 180,E1 -552.201,E2 -552.201} C_VEL
LIN {X 0,Y 601.403,Z 228.571,A -85,B 0,C 180,E1 -552.389,E2 -552.389} C_VEL
LIN {X 0,Y 601.424,Z 228.564,A -85,B 0,C 180,E1 -554.896,E2 -554.896} C_VEL
LIN {X 0,Y 601.424,Z 228.564,A -85,B 0,C 180,E1 -556.985,E2 -556.985} C_VEL
LIN {X 0,Y 601.401,Z 228.574,A -85,B 0,C 180,E1 -559.809,E2 -559.809} C_VEL
LIN {X 0,Y 601.401,Z 228.567,A -85,B 0,C 180,E1 -562.682,E2 -562.682} C_VEL
LIN {X 0,Y 601.398,Z 228.567,A -85,B 0,C 180,E1 -564.878,E2 -564.878} C_VEL
LIN {X 0,Y 601.409,Z 228.571,A -85,B 0,C 180,E1 -567.364,E2 -567.364} C_VEL
LIN {X 0,Y 601.435,Z 228.563,A -85,B 0,C 180,E1 -570.162,E2 -570.162} C_VEL
LIN {X 0,Y 601.418,Z 228.565,A -85,B 0,C 180,E1 -572.717,E2 -572.717} C_VEL
LIN {X 0,Y 601.406,Z 228.573,A -85,B 0,C 180,E1 -575.115,E2 -575.115} C_VEL
LIN {X 0,Y 601.425,Z 228.57,A -85,B 0,C 180,E1 -577.418,E2 -577.418} C_VEL
LIN {X 0,Y 601.402,Z 228.566,A -85,B 0,C 180,E1 -579.994,E2 -579.994} C_VEL
LIN {X 0,Y 601.436,Z 228.567,A -85,B 0,C 180,E1 -582.667,E2 -582.667} C_VEL
LIN {X 0,Y 601.411,Z 228.566,A -85,B 0,C 180,E1 -585.482,E2 -585.482} C_VEL
LIN {X 0,Y 601.418,Z 228.569,A -85,B 0,C 180,E1 -588.406,E2 -588.406} C_VEL
LIN {X 0,Y 601.421,Z 228.569,A -85,B 0,C 180,E1 -590.875,E2 -590.875} C_VEL
LIN {X 0,Y 601.428,Z 228.564,A -85,B 0,C 180,E1 -593.734,E2 -593.734} C_VEL
LIN {X 0,Y 601.417,Z 228.569,A -85,B 0,C 180,E1 -596.687,E2 -596.687} C_VEL
LIN {X 0,Y 601.438,Z 228.566,A -85,B 0,C 180,E1 -599.848,E2 -599.848} C_VEL
LIN {X 0,Y 601.375,Z 228.572,A -85,B 0,C 180,E1 -602.642,E2 -602.642} C_VEL
LIN {X 0,Y 601.377,Z 228.57,A -85,B 0,C 180,E1 -605.121,E2 -605.121} C_VEL
LIN {X 0,Y 601.402,Z 228.569,A -85,B 0,C 180,E1 -607.394,E2 -607.394} C_VEL
LIN {X 0,Y 601.367,Z 229.119,A -85,B 0,C 180,E1 -608.04,E2 -608.04} C_VEL
LIN {X 0,Y 601.387,Z 232.836,A -85,B 0,C 180,E1 -610.19,E2 -610.19} C_VEL
LIN {X 0,Y 601.392,Z 237.772,A -85,B 0,C 180,E1 -613.013,E2 -613.013} C_VEL
LIN {X 0,Y 601.384,Z 242.949,A -85,B 0,C 180,E1 -615.917,E2 -615.917} C_VEL
LIN {X 0,Y 601.366,Z 248.71,A -85,B 0,C 180,E1 -619.01,E2 -619.01} C_VEL
LIN {X 0,Y 601.353,Z 254.295,A -85,B 0,C 180,E1 -621.938,E2 -621.938} C_VEL
LIN {X 0,Y 601.34,Z 259.536,A -85,B 0,C 180,E1 -624.635,E2 -624.635} C_VEL
LIN {X 0,Y 601.333,Z 264.837,A -85,B 0,C 180,E1 -627.321,E2 -627.321} C_VEL
LIN {X 0,Y 601.33,Z 270.196,A -85,B 0,C 180,E1 -630,E2 -630} C_VEL
LIN {X 0,Y 601.345,Z 272.558,A -85,B 0,C 180,E1 -631.172,E2 -631.172} C_VEL
LIN {X 0,Y 601.585,Z 284.057,A -85,B 0,C 180,E1 -631.422,E2 -631.422} C_VEL
LIN {X 0,Y 601.501,Z 297.159,A -85,B 0,C 180,E1 -631.841,E2 -631.841} C_VEL
LIN {X 0,Y 601.489,Z 308.684,A -85,B 0,C 180,E1 -632.344,E2 -632.344} C_VEL
LIN {X 0,Y 601.486,Z 320.584,A -85,B 0,C 180,E1 -633.014,E2 -633.014} C_VEL
LIN {X 0,Y 601.472,Z 331.146,A -85,B 0,C 180,E1 -633.768,E2 -633.768} C_VEL
LIN {X 0,Y 601.415,Z 341.593,A -85,B 0,C 180,E1 -634.692,E2 -634.692} C_VEL
LIN {X 0,Y 601.39,Z 350.665,A -85,B 0,C 180,E1 -635.701,E2 -635.701} C_VEL
LIN {X 0,Y 601.397,Z 358.004,A -85,B 0,C 180,E1 -636.711,E2 -636.711} C_VEL
LIN {X 0,Y 601.374,Z 363.912,A -85,B 0,C 180,E1 -637.723,E2 -637.723} C_VEL
LIN {X 0,Y 601.346,Z 368.584,A -85,B 0,C 180,E1 -638.739,E2 -638.739} C_VEL
LIN {X 0,Y 601.337,Z 372.15,A -85,B 0,C 180,E1 -639.756,E2 -639.756} C_VEL
LIN {X 0,Y 601.349,Z 375.111,A -85,B 0,C 180,E1 -640.981,E2 -640.981} C_VEL
LIN {X 0,Y 601.339,Z 376.623,A -85,B 0,C 180,E1 -642.144,E2 -642.144} C_VEL
LIN {X 0,Y 601.336,Z 376.896,A -85,B 0,C 180,E1 -643.517,E2 -643.517} C_VEL
LIN {X 0,Y 601.314,Z 376.39,A -85,B 0,C 180,E1 -644.208,E2 -644.208} C_VEL
LIN {X 0,Y 601.314,Z 375.456,A -85,B 0,C 180,E1 -644.899,E2 -644.899} C_VEL
LIN {X 0,Y 601.324,Z 374.105,A -85,B 0,C 180,E1 -645.593,E2 -645.593} C_VEL
LIN {X 0,Y 601.333,Z 371.322,A -85,B 0,C 180,E1 -646.596,E2 -646.596} C_VEL
LIN {X 0,Y 601.346,Z 367.154,A -85,B 0,C 180,E1 -647.689,E2 -647.689} C_VEL
LIN {X 0,Y 601.391,Z 361.468,A -85,B 0,C 180,E1 -648.815,E2 -648.815} C_VEL
LIN {X 0,Y 601.371,Z 355.078,A -85,B 0,C 180,E1 -649.81,E2 -649.81} C_VEL
LIN {X 0,Y 601.406,Z 347.236,A -85,B 0,C 180,E1 -650.796,E2 -650.796} C_VEL
LIN {X 0,Y 601.428,Z 337.593,A -85,B 0,C 180,E1 -651.778,E2 -651.778} C_VEL
LIN {X 0,Y 601.45,Z 327.279,A -85,B 0,C 180,E1 -652.616,E2 -652.616} C_VEL
LIN {X 0,Y 601.443,Z 316.63,A -85,B 0,C 180,E1 -653.318,E2 -653.318} C_VEL
LIN {X 0,Y 601.48,Z 306.271,A -85,B 0,C 180,E1 -653.864,E2 -653.864} C_VEL
LIN {X 0,Y 601.54,Z 294.271,A -85,B 0,C 180,E1 -654.356,E2 -654.356} C_VEL
LIN {X 0,Y 601.617,Z 281.248,A -85,B 0,C 180,E1 -654.735,E2 -654.735} C_VEL
LIN {X 0,Y 601.348,Z 273.063,A -85,B 0,C 180,E1 -654.909,E2 -654.909} C_VEL
LIN {X 0,Y 601.297,Z 272.539,A -85,B 0,C 180,E1 -654.929,E2 -654.929} C_VEL
LIN {X 0,Y 601.31,Z 266.626,A -85,B 0,C 180,E1 -657.872,E2 -657.872} C_VEL
LIN {X 0,Y 601.333,Z 262.066,A -85,B 0,C 180,E1 -660.168,E2 -660.168} C_VEL
LIN {X 0,Y 601.331,Z 257.098,A -85,B 0,C 180,E1 -662.704,E2 -662.704} C_VEL
LIN {X 0,Y 601.308,Z 252.473,A -85,B 0,C 180,E1 -665.102,E2 -665.102} C_VEL
LIN {X 0,Y 601.312,Z 248.062,A -85,B 0,C 180,E1 -667.427,E2 -667.427} C_VEL
LIN {X 0,Y 601.348,Z 243.272,A -85,B 0,C 180,E1 -669.999,E2 -669.999} C_VEL
LIN {X 0,Y 601.351,Z 238.508,A -85,B 0,C 180,E1 -672.674,E2 -672.674} C_VEL
LIN {X 0,Y 601.411,Z 233.574,A -85,B 0,C 180,E1 -675.482,E2 -675.482} C_VEL
LIN {X 0,Y 601.38,Z 228.819,A -85,B 0,C 180,E1 -678.233,E2 -678.233} C_VEL
LIN {X 0,Y 601.402,Z 228.571,A -85,B 0,C 180,E1 -679.126,E2 -679.126} C_VEL
LIN {X 0,Y 601.409,Z 228.57,A -85,B 0,C 180,E1 -681.733,E2 -681.733} C_VEL
LIN {X 0,Y 601.401,Z 228.577,A -85,B 0,C 180,E1 -684.248,E2 -684.248} C_VEL
LIN {X 0,Y 601.398,Z 228.571,A -85,B 0,C 180,E1 -686.686,E2 -686.686} C_VEL
LIN {X 0,Y 601.424,Z 228.57,A -85,B 0,C 180,E1 -689.06,E2 -689.06} C_VEL
LIN {X 0,Y 601.433,Z 228.567,A -85,B 0,C 180,E1 -691.374,E2 -691.374} C_VEL
LIN {X 0,Y 601.385,Z 228.572,A -85,B 0,C 180,E1 -694.135,E2 -694.135} C_VEL
LIN {X 0,Y 601.417,Z 228.571,A -85,B 0,C 180,E1 -696.591,E2 -696.591} C_VEL
LIN {X 0,Y 601.421,Z 228.572,A -85,B 0,C 180,E1 -699.479,E2 -699.479} C_VEL
LIN {X 0,Y 601.387,Z 228.577,A -85,B 0,C 180,E1 -702.312,E2 -702.312} C_VEL
LIN {X 0,Y 601.414,Z 228.569,A -85,B 0,C 180,E1 -704.41,E2 -704.41} C_VEL
LIN {X 0,Y 601.399,Z 228.573,A -85,B 0,C 180,E1 -707.172,E2 -707.172} C_VEL
LIN {X 0,Y 601.429,Z 228.573,A -85,B 0,C 180,E1 -709.906,E2 -709.906} C_VEL
LIN {X 0,Y 601.446,Z 228.567,A -85,B 0,C 180,E1 -712.616,E2 -712.616} C_VEL
LIN {X 0,Y 601.402,Z 228.57,A -85,B 0,C 180,E1 -715.309,E2 -715.309} C_VEL
LIN {X 0,Y 601.413,Z 228.569,A -85,B 0,C 180,E1 -717.992,E2 -717.992} C_VEL
LIN {X 0,Y 601.44,Z 228.569,A -85,B 0,C 180,E1 -720.67,E2 -720.67} C_VEL
LIN {X 0,Y 601.426,Z 228.571,A -85,B 0,C 180,E1 -723.35,E2 -723.35} C_VEL
LIN {X 0,Y 601.396,Z 228.572,A -85,B 0,C 180,E1 -726.038,E2 -726.038} C_VEL
LIN {X 0,Y 601.404,Z 228.57,A -85,B 0,C 180,E1 -728.739,E2 -728.739} C_VEL
LIN {X 0,Y 601.429,Z 228.568,A -85,B 0,C 180,E1 -731.459,E2 -731.459} C_VEL
LIN {X 0,Y 601.404,Z 228.574,A -85,B 0,C 180,E1 -734.206,E2 -734.206} C_VEL
LIN {X 0,Y 601.426,Z 228.572,A -85,B 0,C 180,E1 -736.987,E2 -736.987} C_VEL
LIN {X 0,Y 601.394,Z 228.574,A -85,B 0,C 180,E1 -739.81,E2 -739.81} C_VEL
LIN {X 0,Y 601.404,Z 228.571,A -85,B 0,C 180,E1 -742.684,E2 -742.684} C_VEL
LIN {X 0,Y 601.395,Z 228.574,A -85,B 0,C 180,E1 -744.88,E2 -744.88} C_VEL
LIN {X 0,Y 601.395,Z 228.574,A -85,B 0,C 180,E1 -747.361,E2 -747.361} C_VEL
LIN {X 0,Y 601.422,Z 228.569,A -85,B 0,C 180,E1 -750.165,E2 -750.165} C_VEL
LIN {X 0,Y 601.409,Z 228.57,A -85,B 0,C 180,E1 -752.716,E2 -752.716} C_VEL
LIN {X 0,Y 601.384,Z 228.577,A -85,B 0,C 180,E1 -755.112,E2 -755.112} C_VEL
LIN {X 0,Y 601.433,Z 228.566,A -85,B 0,C 180,E1 -757.42,E2 -757.42} C_VEL
LIN {X 0,Y 601.407,Z 228.572,A -85,B 0,C 180,E1 -759.996,E2 -759.996} C_VEL
LIN {X 0,Y 601.404,Z 228.575,A -85,B 0,C 180,E1 -762.671,E2 -762.671} C_VEL
LIN {X 0,Y 601.423,Z 228.57,A -85,B 0,C 180,E1 -765.483,E2 -765.483} C_VEL
LIN {X 0,Y 601.412,Z 228.571,A -85,B 0,C 180,E1 -768.409,E2 -768.409} C_VEL
LIN {X 0,Y 601.439,Z 228.566,A -85,B 0,C 180,E1 -770.877,E2 -770.877} C_VEL
LIN {X 0,Y 601.402,Z 228.576,A -85,B 0,C 180,E1 -773.418,E2 -773.418} C_VEL
LIN {X 0,Y 601.432,Z 228.72,A -85,B 0,C 180,E1 -774.336,E2 -774.336} C_VEL
LIN {X 0,Y 601.526,Z 235.095,A -85,B 0,C 180,E1 -776.694,E2 -776.694} C_VEL
LIN {X 0,Y 601.472,Z 242.852,A -85,B 0,C 180,E1 -779.451,E2 -779.451} C_VEL
LIN {X 0,Y 601.425,Z 250.754,A -85,B 0,C 180,E1 -782.134,E2 -782.134} C_VEL
LIN {X 0,Y 601.413,Z 259.658,A -85,B 0,C 180,E1 -785.123,E2 -785.123} C_VEL
LIN {X 0,Y 601.417,Z 266.574,A -85,B 0,C 180,E1 -787.395,E2 -787.395} C_VEL
LIN {X 0,Y 601.413,Z 275.241,A -85,B 0,C 180,E1 -790.191,E2 -790.191} C_VEL
LIN {X 0,Y 601.376,Z 284.145,A -85,B 0,C 180,E1 -793.013,E2 -793.013} C_VEL
LIN {X 0,Y 601.355,Z 293.049,A -85,B 0,C 180,E1 -795.793,E2 -795.793} C_VEL
LIN {X 0,Y 601.371,Z 300.493,A -85,B 0,C 180,E1 -798.092,E2 -798.092} C_VEL
LIN {X 0,Y 601.607,Z 307.528,A -85,B 0,C 180,E1 -798.225,E2 -798.225} C_VEL
LIN {X 0,Y 601.555,Z 319.888,A -85,B 0,C 180,E1 -798.545,E2 -798.545} C_VEL
LIN {X 0,Y 601.492,Z 332.869,A -85,B 0,C 180,E1 -799.028,E2 -799.028} C_VEL
LIN {X 0,Y 601.449,Z 345.332,A -85,B 0,C 180,E1 -799.65,E2 -799.65} C_VEL
LIN {X 0,Y 601.464,Z 355.935,A -85,B 0,C 180,E1 -800.33,E2 -800.33} C_VEL
LIN {X 0,Y 601.435,Z 365.602,A -85,B 0,C 180,E1 -801.093,E2 -801.093} C_VEL
LIN {X 0,Y 601.406,Z 374.415,A -85,B 0,C 180,E1 -801.939,E2 -801.939} C_VEL
LIN {X 0,Y 601.388,Z 381.692,A -85,B 0,C 180,E1 -802.783,E2 -802.783} C_VEL
LIN {X 0,Y 601.375,Z 388.775,A -85,B 0,C 180,E1 -803.782,E2 -803.782} C_VEL
LIN {X 0,Y 601.373,Z 393.681,A -85,B 0,C 180,E1 -804.636,E2 -804.636} C_VEL
LIN {X 0,Y 601.354,Z 398.372,A -85,B 0,C 180,E1 -805.643,E2 -805.643} C_VEL
LIN {X 0,Y 601.344,Z 401.956,A -85,B 0,C 180,E1 -806.65,E2 -806.65} C_VEL
LIN {X 0,Y 601.325,Z 403.809,A -85,B 0,C 180,E1 -807.321,E2 -807.321} C_VEL
LIN {X 0,Y 601.343,Z 405.202,A -85,B 0,C 180,E1 -807.991,E2 -807.991} C_VEL
LIN {X 0,Y 601.339,Z 406.784,A -85,B 0,C 180,E1 -809.33,E2 -809.33} C_VEL
LIN {X 0,Y 601.335,Z 407,A -85,B 0,C 180,E1 -810,E2 -810} C_VEL
LIN {X 0,Y 601.347,Z 406.184,A -85,B 0,C 180,E1 -811.339,E2 -811.339} C_VEL
LIN {X 0,Y 601.343,Z 405.202,A -85,B 0,C 180,E1 -812.009,E2 -812.009} C_VEL
LIN {X 0,Y 601.325,Z 403.809,A -85,B 0,C 180,E1 -812.68,E2 -812.68} C_VEL
LIN {X 0,Y 601.368,Z 400.896,A -85,B 0,C 180,E1 -813.685,E2 -813.685} C_VEL
LIN {X 0,Y 601.336,Z 396.95,A -85,B 0,C 180,E1 -814.693,E2 -814.693} C_VEL
LIN {X 0,Y 601.373,Z 390.878,A -85,B 0,C 180,E1 -815.869,E2 -815.869} C_VEL
LIN {X 0,Y 601.382,Z 384.237,A -85,B 0,C 180,E1 -816.88,E2 -816.88} C_VEL
LIN {X 0,Y 601.4,Z 375.991,A -85,B 0,C 180,E1 -817.892,E2 -817.892} C_VEL
LIN {X 0,Y 601.436,Z 367.539,A -85,B 0,C 180,E1 -818.737,E2 -818.737} C_VEL
LIN {X 0,Y 601.447,Z 357.095,A -85,B 0,C 180,E1 -819.585,E2 -819.585} C_VEL
LIN {X 0,Y 601.473,Z 346.761,A -85,B 0,C 180,E1 -820.264,E2 -820.264} C_VEL
LIN {X 0,Y 601.481,Z 335.255,A -85,B 0,C 180,E1 -820.868,E2 -820.868} C_VEL
LIN {X 0,Y 601.526,Z 322.346,A -85,B 0,C 180,E1 -821.375,E2 -821.375} C_VEL
LIN {X 0,Y 601.611,Z 309.448,A -85,B 0,C 180,E1 -821.732,E2 -821.732} C_VEL
LIN {X 0,Y 601.501,Z 301.631,A -85,B 0,C 180,E1 -821.884,E2 -821.884} C_VEL
LIN {X 0,Y 601.342,Z 300.423,A -85,B 0,C 180,E1 -821.93,E2 -821.93} C_VEL
LIN {X 0,Y 601.352,Z 291.936,A -85,B 0,C 180,E1 -824.552,E2 -824.552} C_VEL
LIN {X 0,Y 601.394,Z 283.032,A -85,B 0,C 180,E1 -827.337,E2 -827.337} C_VEL
LIN {X 0,Y 601.394,Z 274.128,A -85,B 0,C 180,E1 -830.166,E2 -830.166} C_VEL
LIN {X 0,Y 601.412,Z 266.336,A -85,B 0,C 180,E1 -832.682,E2 -832.682} C_VEL
LIN {X 0,Y 601.409,Z 258.545,A -85,B 0,C 180,E1 -835.247,E2 -835.247} C_VEL
LIN {X 0,Y 601.425,Z 250.753,A -85,B 0,C 180,E1 -837.866,E2 -837.866} C_VEL
LIN {X 0,Y 601.472,Z 242.888,A -85,B 0,C 180,E1 -840.549,E2 -840.549} C_VEL
LIN {X 0,Y 601.526,Z 235.103,A -85,B 0,C 180,E1 -843.306,E2 -843.306} C_VEL
LIN {X 0,Y 601.409,Z 228.606,A -85,B 0,C 180,E1 -845.709,E2 -845.709} C_VEL
LIN {X 0,Y 601.39,Z 228.57,A -85,B 0,C 180,E1 -848.465,E2 -848.465} C_VEL
LIN {X 0,Y 601.396,Z 228.577,A -85,B 0,C 180,E1 -850.875,E2 -850.875} C_VEL
LIN {X 0,Y 601.395,Z 228.568,A -85,B 0,C 180,E1 -853.588,E2 -853.588} C_VEL
LIN {X 0,Y 601.402,Z 228.572,A -85,B 0,C 180,E1 -856.429,E2 -856.429} C_VEL
LIN {X 0,Y 601.39,Z 228.57,A -85,B 0,C 180,E1 -859.123,E2 -859.123} C_VEL
LIN {X 0,Y 601.353,Z 228.573,A -85,B 0,C 180,E1 -861.726,E2 -861.726} C_VEL
LIN {X 0,Y 601.375,Z 228.578,A -85,B 0,C 180,E1 -864.244,E2 -864.244} C_VEL
LIN {X 0,Y 601.411,Z 228.568,A -85,B 0,C 180,E1 -866.685,E2 -866.685} C_VEL
LIN {X 0,Y 601.385,Z 228.569,A -85,B 0,C 180,E1 -869.055,E2 -869.055} C_VEL
LIN {X 0,Y 601.394,Z 228.569,A -85,B 0,C 180,E1 -871.371,E2 -871.371} C_VEL
LIN {X 0,Y 601.407,Z 228.569,A -85,B 0,C 180,E1 -874.381,E2 -874.381} C_VEL
LIN {X 0,Y 601.381,Z 228.569,A -85,B 0,C 180,E1 -876.587,E2 -876.587} C_VEL
LIN {X 0,Y 601.419,Z 228.571,A -85,B 0,C 180,E1 -879.477,E2 -879.477} C_VEL
LIN {X 0,Y 601.381,Z 228.57,A -85,B 0,C 180,E1 -882.311,E2 -882.311} C_VEL
LIN {X 0,Y 601.395,Z 228.567,A -85,B 0,C 180,E1 -884.408,E2 -884.408} C_VEL
LIN {X 0,Y 601.413,Z 228.572,A -85,B 0,C 180,E1 -887.171,E2 -887.171} C_VEL
LIN {X 0,Y 601.422,Z 228.565,A -85,B 0,C 180,E1 -889.904,E2 -889.904} C_VEL
LIN {X 0,Y 601.427,Z 228.566,A -85,B 0,C 180,E1 -892.614,E2 -892.614} C_VEL
LIN {X 0,Y 601.425,Z 228.569,A -85,B 0,C 180,E1 -895.307,E2 -895.307} C_VEL
LIN {X 0,Y 601.407,Z 228.566,A -85,B 0,C 180,E1 -897.99,E2 -897.99} C_VEL
LIN {X 0,Y 601.451,Z 228.569,A -85,B 0,C 180,E1 -900.669,E2 -900.669} C_VEL
LIN {X 0,Y 601.43,Z 228.564,A -85,B 0,C 180,E1 -903.349,E2 -903.349} C_VEL
LIN {X 0,Y 601.399,Z 228.569,A -85,B 0,C 180,E1 -906.036,E2 -906.036} C_VEL
LIN {X 0,Y 601.437,Z 228.567,A -85,B 0,C 180,E1 -908.737,E2 -908.737} C_VEL
LIN {X 0,Y 601.43,Z 228.563,A -85,B 0,C 180,E1 -911.457,E2 -911.457} C_VEL
LIN {X 0,Y 601.403,Z 228.571,A -85,B 0,C 180,E1 -912.389,E2 -912.389} C_VEL
LIN {X 0,Y 600.743,Z 228.651,A -85,B 0,C 180,E1 -912.948,E2 -912.948} C_VEL
LIN {X 0,Y 597.892,Z 229.008,A -85,B 0,C 180,E1 -913.856,E2 -913.856} C_VEL
LIN {X 0,Y 595.479,Z 229.308,A -85,B 0,C 180,E1 -914.586,E2 -914.586} C_VEL
LIN {X 0,Y 594.442,Z 229.434,A -85,B 0,C 180,E1 -915.15,E2 -915.15} C_VEL
LIN {X 0,Y 594.357,Z 229.445,A -85,B 0,C 180,E1 -915.341,E2 -915.341} C_VEL
LIN {X 0,Y 594.376,Z 229.45,A -85,B 0,C 180,E1 -917.903,E2 -917.903} C_VEL
LIN {X 0,Y 594.372,Z 229.442,A -85,B 0,C 180,E1 -920.918,E2 -920.918} C_VEL
LIN {X 0,Y 594.385,Z 229.45,A -85,B 0,C 180,E1 -923.703,E2 -923.703} C_VEL
LIN {X 0,Y 594.38,Z 229.441,A -85,B 0,C 180,E1 -926.699,E2 -926.699} C_VEL
LIN {X 0,Y 594.375,Z 229.444,A -85,B 0,C 180,E1 -928.998,E2 -928.998} C_VEL
LIN {X 0,Y 594.381,Z 229.447,A -85,B 0,C 180,E1 -931.645,E2 -931.645} C_VEL
LIN {X 0,Y 594.388,Z 229.441,A -85,B 0,C 180,E1 -934.578,E2 -934.578} C_VEL
LIN {X 0,Y 594.377,Z 229.45,A -85,B 0,C 180,E1 -937.086,E2 -937.086} C_VEL
LIN {X 0,Y 594.365,Z 229.444,A -85,B 0,C 180,E1 -939.775,E2 -939.775} C_VEL
LIN {X 0,Y 594.383,Z 229.442,A -85,B 0,C 180,E1 -942.373,E2 -942.373} C_VEL
LIN {X 0,Y 594.349,Z 229.449,A -85,B 0,C 180,E1 -945.191,E2 -945.191} C_VEL
LIN {X 0,Y 594.353,Z 229.444,A -85,B 0,C 180,E1 -947.624,E2 -947.624} C_VEL
LIN {X 0,Y 594.381,Z 229.446,A -85,B 0,C 180,E1 -950.321,E2 -950.321} C_VEL
LIN {X 0,Y 594.369,Z 229.446,A -85,B 0,C 180,E1 -952.913,E2 -952.913} C_VEL
LIN {X 0,Y 594.37,Z 229.445,A -85,B 0,C 180,E1 -955.861,E2 -955.861} C_VEL
LIN {X 0,Y 594.354,Z 229.448,A -85,B 0,C 180,E1 -958.65,E2 -958.65} C_VEL
LIN {X 0,Y 594.364,Z 229.443,A -85,B 0,C 180,E1 -961.043,E2 -961.043} C_VEL
LIN {X 0,Y 594.355,Z 229.454,A -85,B 0,C 180,E1 -964.056,E2 -964.056} C_VEL
LIN {X 0,Y 594.365,Z 229.447,A -85,B 0,C 180,E1 -966.296,E2 -966.296} C_VEL
LIN {X 0,Y 594.326,Z 229.482,A -85,B 0,C 180,E1 -967.766,E2 -967.766} C_VEL
LIN {X 0,Y 594.333,Z 233.196,A -85,B 0,C 180,E1 -969.945,E2 -969.945} C_VEL
LIN {X 0,Y 594.337,Z 238.151,A -85,B 0,C 180,E1 -972.805,E2 -972.805} C_VEL
LIN {X 0,Y 594.323,Z 243.524,A -85,B 0,C 180,E1 -975.847,E2 -975.847} C_VEL
LIN {X 0,Y 594.283,Z 248.148,A -85,B 0,C 180,E1 -978.402,E2 -978.402} C_VEL
LIN {X 0,Y 594.308,Z 253.31,A -85,B 0,C 180,E1 -981.157,E2 -981.157} C_VEL
LIN {X 0,Y 594.26,Z 258.537,A -85,B 0,C 180,E1 -983.89,E2 -983.89} C_VEL
LIN {X 0,Y 594.242,Z 262.495,A -85,B 0,C 180,E1 -985.931,E2 -985.931} C_VEL
LIN {X 0,Y 594.238,Z 267.824,A -85,B 0,C 180,E1 -988.645,E2 -988.645} C_VEL
LIN {X 0,Y 594.267,Z 272.535,A -85,B 0,C 180,E1 -991.016,E2 -991.016} C_VEL
LIN {X 0,Y 594.669,Z 278.103,A -85,B 0,C 180,E1 -991.143,E2 -991.143} C_VEL
LIN {X 0,Y 594.585,Z 290.733,A -85,B 0,C 180,E1 -991.482,E2 -991.482} C_VEL
LIN {X 0,Y 594.5,Z 302.982,A -85,B 0,C 180,E1 -991.948,E2 -991.948} C_VEL
LIN {X 0,Y 594.496,Z 314.762,A -85,B 0,C 180,E1 -992.541,E2 -992.541} C_VEL
LIN {X 0,Y 594.469,Z 325.367,A -85,B 0,C 180,E1 -993.219,E2 -993.219} C_VEL
LIN {X 0,Y 594.391,Z 336.012,A -85,B 0,C 180,E1 -994.068,E2 -994.068} C_VEL
LIN {X 0,Y 594.354,Z 344.701,A -85,B 0,C 180,E1 -994.918,E2 -994.918} C_VEL
LIN {X 0,Y 594.323,Z 353.191,A -85,B 0,C 180,E1 -995.939,E2 -995.939} C_VEL
LIN {X 0,Y 594.299,Z 360.025,A -85,B 0,C 180,E1 -996.962,E2 -996.962} C_VEL
LIN {X 0,Y 594.276,Z 366.323,A -85,B 0,C 180,E1 -998.158,E2 -998.158} C_VEL
LIN {X 0,Y 594.26,Z 370.444,A -85,B 0,C 180,E1 -999.187,E2 -999.187} C_VEL
LIN {X 0,Y 594.23,Z 373.512,A -85,B 0,C 180,E1 -1000.218,E2 -1000.218} C_VEL
LIN {X 0,Y 594.267,Z 375.214,A -85,B 0,C 180,E1 -1001.02,E2 -1001.02} C_VEL
LIN {X 0,Y 594.235,Z 376.732,A -85,B 0,C 180,E1 -1002.291,E2 -1002.291} C_VEL
LIN {X 0,Y 594.24,Z 376.992,A -85,B 0,C 180,E1 -1002.986,E2 -1002.986} C_VEL
LIN {X 0,Y 594.248,Z 376.497,A -85,B 0,C 180,E1 -1004.125,E2 -1004.125} C_VEL
LIN {X 0,Y 594.224,Z 375.196,A -85,B 0,C 180,E1 -1005.081,E2 -1005.081} C_VEL
LIN {X 0,Y 594.25,Z 373.74,A -85,B 0,C 180,E1 -1005.784,E2 -1005.784} C_VEL
LIN {X 0,Y 594.245,Z 371.207,A -85,B 0,C 180,E1 -1006.675,E2 -1006.675} C_VEL
LIN {X 0,Y 594.262,Z 366.439,A -85,B 0,C 180,E1 -1007.907,E2 -1007.907} C_VEL
LIN {X 0,Y 594.317,Z 360.279,A -85,B 0,C 180,E1 -1009.085,E2 -1009.085} C_VEL
LIN {X 0,Y 594.312,Z 352.573,A -85,B 0,C 180,E1 -1010.236,E2 -1010.236} C_VEL
LIN {X 0,Y 594.381,Z 344.751,A -85,B 0,C 180,E1 -1011.167,E2 -1011.167} C_VEL
LIN {X 0,Y 594.421,Z 334.681,A -85,B 0,C 180,E1 -1012.139,E2 -1012.139} C_VEL
LIN {X 0,Y 594.452,Z 324.054,A -85,B 0,C 180,E1 -1012.963,E2 -1012.963} C_VEL
LIN {X 0,Y 594.449,Z 312.019,A -85,B 0,C 180,E1 -1013.701,E2 -1013.701} C_VEL
LIN {X 0,Y 594.527,Z 300.425,A -85,B 0,C 180,E1 -1014.254,E2 -1014.254} C_VEL
LIN {X 0,Y 594.652,Z 287.628,A -85,B 0,C 180,E1 -1014.704,E2 -1014.704} C_VEL
LIN {X 0,Y 594.457,Z 274.161,A -85,B 0,C 180,E1 -1015.027,E2 -1015.027} C_VEL
LIN {X 0,Y 594.201,Z 272.541,A -85,B 0,C 180,E1 -1015.072,E2 -1015.072} C_VEL
LIN {X 0,Y 594.21,Z 267.724,A -85,B 0,C 180,E1 -1017.497,E2 -1017.497} C_VEL
LIN {X 0,Y 594.232,Z 262.211,A -85,B 0,C 180,E1 -1020.305,E2 -1020.305} C_VEL
LIN {X 0,Y 594.237,Z 257.08,A -85,B 0,C 180,E1 -1022.958,E2 -1022.958} C_VEL
LIN {X 0,Y 594.241,Z 252.403,A -85,B 0,C 180,E1 -1025.415,E2 -1025.415} C_VEL
LIN {X 0,Y 594.252,Z 247.665,A -85,B 0,C 180,E1 -1027.95,E2 -1027.95} C_VEL
LIN {X 0,Y 594.261,Z 242.96,A -85,B 0,C 180,E1 -1030.575,E2 -1030.575} C_VEL
LIN {X 0,Y 594.325,Z 238.15,A -85,B 0,C 180,E1 -1033.302,E2 -1033.302} C_VEL
LIN {X 0,Y 594.356,Z 233.17,A -85,B 0,C 180,E1 -1036.16,E2 -1036.16} C_VEL
LIN {X 0,Y 594.344,Z 229.785,A -85,B 0,C 180,E1 -1038.154,E2 -1038.154} C_VEL
LIN {X 0,Y 594.339,Z 229.453,A -85,B 0,C 180,E1 -1038.534,E2 -1038.534} C_VEL
LIN {X 0,Y 594.369,Z 229.452,A -85,B 0,C 180,E1 -1041.296,E2 -1041.296} C_VEL
LIN {X 0,Y 594.387,Z 229.445,A -85,B 0,C 180,E1 -1043.759,E2 -1043.759} C_VEL
LIN {X 0,Y 594.349,Z 229.45,A -85,B 0,C 180,E1 -1046.238,E2 -1046.238} C_VEL
LIN {X 0,Y 594.379,Z 229.45,A -85,B 0,C 180,E1 -1048.652,E2 -1048.652} C_VEL
LIN {X 0,Y 594.381,Z 229.445,A -85,B 0,C 180,E1 -1051.04,E2 -1051.04} C_VEL
LIN {X 0,Y 594.361,Z 229.447,A -85,B 0,C 180,E1 -1053.979,E2 -1053.979} C_VEL
LIN {X 0,Y 594.382,Z 229.45,A -85,B 0,C 180,E1 -1056.297,E2 -1056.297} C_VEL
LIN {X 0,Y 594.398,Z 229.447,A -85,B 0,C 180,E1 -1059.225,E2 -1059.225} C_VEL
LIN {X 0,Y 594.366,Z 229.449,A -85,B 0,C 180,E1 -1062.096,E2 -1062.096} C_VEL
LIN {X 0,Y 594.366,Z 229.449,A -85,B 0,C 180,E1 -1064.22,E2 -1064.22} C_VEL
LIN {X 0,Y 594.348,Z 229.454,A -85,B 0,C 180,E1 -1067.018,E2 -1067.018} C_VEL
LIN {X 0,Y 594.387,Z 229.448,A -85,B 0,C 180,E1 -1069.785,E2 -1069.785} C_VEL
LIN {X 0,Y 594.393,Z 229.445,A -85,B 0,C 180,E1 -1072.528,E2 -1072.528} C_VEL
LIN {X 0,Y 594.374,Z 229.446,A -85,B 0,C 180,E1 -1075.253,E2 -1075.253} C_VEL
LIN {X 0,Y 594.384,Z 229.445,A -85,B 0,C 180,E1 -1077.968,E2 -1077.968} C_VEL
LIN {X 0,Y 594.411,Z 229.445,A -85,B 0,C 180,E1 -1080.678,E2 -1080.678} C_VEL
LIN {X 0,Y 594.377,Z 229.45,A -85,B 0,C 180,E1 -1083.39,E2 -1083.39} C_VEL
LIN {X 0,Y 594.351,Z 229.45,A -85,B 0,C 180,E1 -1086.11,E2 -1086.11} C_VEL
LIN {X 0,Y 594.371,Z 229.446,A -85,B 0,C 180,E1 -1088.843,E2 -1088.843} C_VEL
LIN {X 0,Y 594.387,Z 229.444,A -85,B 0,C 180,E1 -1091.597,E2 -1091.597} C_VEL
LIN {X 0,Y 594.373,Z 229.448,A -85,B 0,C 180,E1 -1094.378,E2 -1094.378} C_VEL
LIN {X 0,Y 594.385,Z 229.449,A -85,B 0,C 180,E1 -1097.194,E2 -1097.194} C_VEL
LIN {X 0,Y 594.361,Z 229.453,A -85,B 0,C 180,E1 -1100.055,E2 -1100.055} C_VEL
LIN {X 0,Y 594.358,Z 229.452,A -85,B 0,C 180,E1 -1102.968,E2 -1102.968} C_VEL
LIN {X 0,Y 594.371,Z 229.447,A -85,B 0,C 180,E1 -1105.194,E2 -1105.194} C_VEL
LIN {X 0,Y 594.342,Z 229.454,A -85,B 0,C 180,E1 -1107.521,E2 -1107.521} C_VEL
LIN {X 0,Y 594.382,Z 229.447,A -85,B 0,C 180,E1 -1110.33,E2 -1110.33} C_VEL
LIN {X 0,Y 594.371,Z 229.446,A -85,B 0,C 180,E1 -1112.951,E2 -1112.951} C_VEL
LIN {X 0,Y 594.343,Z 229.453,A -85,B 0,C 180,E1 -1115.41,E2 -1115.41} C_VEL
LIN {X 0,Y 594.385,Z 229.447,A -85,B 0,C 180,E1 -1117.941,E2 -1117.941} C_VEL
LIN {X 0,Y 594.366,Z 229.448,A -85,B 0,C 180,E1 -1120.822,E2 -1120.822} C_VEL
LIN {X 0,Y 594.38,Z 229.446,A -85,B 0,C 180,E1 -1123.842,E2 -1123.842} C_VEL
LIN {X 0,Y 594.342,Z 229.451,A -85,B 0,C 180,E1 -1126.7,E2 -1126.7} C_VEL
LIN {X 0,Y 594.361,Z 229.448,A -85,B 0,C 180,E1 -1129.434,E2 -1129.434} C_VEL
LIN {X 0,Y 594.388,Z 229.448,A -85,B 0,C 180,E1 -1132.06,E2 -1132.06} C_VEL
LIN {X 0,Y 594.371,Z 229.586,A -85,B 0,C 180,E1 -1134.177,E2 -1134.177} C_VEL
LIN {X 0,Y 594.477,Z 233.981,A -85,B 0,C 180,E1 -1135.849,E2 -1135.849} C_VEL
LIN {X 0,Y 594.474,Z 239.492,A -85,B 0,C 180,E1 -1137.86,E2 -1137.86} C_VEL
LIN {X 0,Y 594.438,Z 247.281,A -85,B 0,C 180,E1 -1140.617,E2 -1140.617} C_VEL
LIN {X 0,Y 594.378,Z 255.203,A -85,B 0,C 180,E1 -1143.301,E2 -1143.301} C_VEL
LIN {X 0,Y 594.41,Z 263.012,A -85,B 0,C 180,E1 -1145.932,E2 -1145.932} C_VEL
LIN {X 0,Y 594.387,Z 270.789,A -85,B 0,C 180,E1 -1148.498,E2 -1148.498} C_VEL
LIN {X 0,Y 594.327,Z 279.693,A -85,B 0,C 180,E1 -1151.381,E2 -1151.381} C_VEL
LIN {X 0,Y 594.301,Z 288.597,A -85,B 0,C 180,E1 -1154.218,E2 -1154.218} C_VEL
LIN {X 0,Y 594.276,Z 297.501,A -85,B 0,C 180,E1 -1157.015,E2 -1157.015} C_VEL
LIN {X 0,Y 594.28,Z 300.493,A -85,B 0,C 180,E1 -1157.948,E2 -1157.948} C_VEL
LIN {X 0,Y 594.668,Z 305.247,A -85,B 0,C 180,E1 -1158.043,E2 -1158.043} C_VEL
LIN {X 0,Y 594.612,Z 318.508,A -85,B 0,C 180,E1 -1158.366,E2 -1158.366} C_VEL
LIN {X 0,Y 594.53,Z 330.683,A -85,B 0,C 180,E1 -1158.803,E2 -1158.803} C_VEL
LIN {X 0,Y 594.472,Z 342.215,A -85,B 0,C 180,E1 -1159.355,E2 -1159.355} C_VEL
LIN {X 0,Y 594.459,Z 353.481,A -85,B 0,C 180,E1 -1160.044,E2 -1160.044} C_VEL
LIN {X 0,Y 594.406,Z 363.65,A -85,B 0,C 180,E1 -1160.816,E2 -1160.816} C_VEL
LIN {X 0,Y 594.372,Z 372.789,A -85,B 0,C 180,E1 -1161.672,E2 -1161.672} C_VEL
LIN {X 0,Y 594.316,Z 381.692,A -85,B 0,C 180,E1 -1162.697,E2 -1162.697} C_VEL
LIN {X 0,Y 594.281,Z 388.171,A -85,B 0,C 180,E1 -1163.615,E2 -1163.615} C_VEL
LIN {X 0,Y 594.289,Z 393.681,A -85,B 0,C 180,E1 -1164.571,E2 -1164.571} C_VEL
LIN {X 0,Y 594.27,Z 398.372,A -85,B 0,C 180,E1 -1165.591,E2 -1165.591} C_VEL
LIN {X 0,Y 594.267,Z 401.957,A -85,B 0,C 180,E1 -1166.61,E2 -1166.61} C_VEL
LIN {X 0,Y 594.226,Z 403.809,A -85,B 0,C 180,E1 -1167.288,E2 -1167.288} C_VEL
LIN {X 0,Y 594.242,Z 405.201,A -85,B 0,C 180,E1 -1167.967,E2 -1167.967} C_VEL
LIN {X 0,Y 594.239,Z 406.784,A -85,B 0,C 180,E1 -1169.322,E2 -1169.322} C_VEL
LIN {X 0,Y 594.236,Z 407,A -85,B 0,C 180,E1 -1170,E2 -1170} C_VEL
LIN {X 0,Y 594.247,Z 406.185,A -85,B 0,C 180,E1 -1171.355,E2 -1171.355} C_VEL
LIN {X 0,Y 594.242,Z 405.202,A -85,B 0,C 180,E1 -1172.033,E2 -1172.033} C_VEL
LIN {X 0,Y 594.226,Z 403.81,A -85,B 0,C 180,E1 -1172.712,E2 -1172.712} C_VEL
LIN {X 0,Y 594.289,Z 400.896,A -85,B 0,C 180,E1 -1173.729,E2 -1173.729} C_VEL
LIN {X 0,Y 594.241,Z 396.95,A -85,B 0,C 180,E1 -1174.749,E2 -1174.749} C_VEL
LIN {X 0,Y 594.305,Z 390.878,A -85,B 0,C 180,E1 -1175.939,E2 -1175.939} C_VEL
LIN {X 0,Y 594.308,Z 384.237,A -85,B 0,C 180,E1 -1176.962,E2 -1176.962} C_VEL
LIN {X 0,Y 594.359,Z 375.991,A -85,B 0,C 180,E1 -1177.986,E2 -1177.986} C_VEL
LIN {X 0,Y 594.382,Z 367.539,A -85,B 0,C 180,E1 -1178.842,E2 -1178.842} C_VEL
LIN {X 0,Y 594.432,Z 357.096,A -85,B 0,C 180,E1 -1179.699,E2 -1179.699} C_VEL
LIN {X 0,Y 594.45,Z 346.763,A -85,B 0,C 180,E1 -1180.387,E2 -1180.387} C_VEL
LIN {X 0,Y 594.499,Z 334.785,A -85,B 0,C 180,E1 -1181.018,E2 -1181.018} C_VEL
LIN {X 0,Y 594.56,Z 322.502,A -85,B 0,C 180,E1 -1181.505,E2 -1181.505} C_VEL
LIN {X 0,Y 594.68,Z 309.447,A -85,B 0,C 180,E1 -1181.871,E2 -1181.871} C_VEL
LIN {X 0,Y 594.419,Z 301.63,A -85,B 0,C 180,E1 -1182.028,E2 -1182.028} C_VEL
LIN {X 0,Y 594.285,Z 300.423,A -85,B 0,C 180,E1 -1182.074,E2 -1182.074} C_VEL
LIN {X 0,Y 594.299,Z 291.936,A -85,B 0,C 180,E1 -1184.729,E2 -1184.729} C_VEL
LIN {X 0,Y 594.325,Z 283.032,A -85,B 0,C 180,E1 -1187.55,E2 -1187.55} C_VEL
LIN {X 0,Y 594.358,Z 274.128,A -85,B 0,C 180,E1 -1190.415,E2 -1190.415} C_VEL
LIN {X 0,Y 594.375,Z 266.336,A -85,B 0,C 180,E1 -1192.966,E2 -1192.966} C_VEL
LIN {X 0,Y 594.407,Z 258.545,A -85,B 0,C 180,E1 -1195.566,E2 -1195.566} C_VEL
LIN {X 0,Y 594.384,Z 250.658,A -85,B 0,C 180,E1 -1198.226,E2 -1198.226} C_VEL
LIN {X 0,Y 594.467,Z 242.844,A -85,B 0,C 180,E1 -1200.948,E2 -1200.948} C_VEL
LIN {X 0,Y 594.511,Z 235.086,A -85,B 0,C 180,E1 -1203.752,E2 -1203.752} C_VEL
LIN {X 0,Y 594.545,Z 230.689,A -85,B 0,C 180,E1 -1205.395,E2 -1205.395} C_VEL
LIN {X 0,Y 594.348,Z 229.452,A -85,B 0,C 180,E1 -1205.929,E2 -1205.929} C_VEL
LIN {X 0,Y 594.359,Z 229.449,A -85,B 0,C 180,E1 -1208.701,E2 -1208.701} C_VEL
LIN {X 0,Y 594.341,Z 229.448,A -85,B 0,C 180,E1 -1211.466,E2 -1211.466} C_VEL
LIN {X 0,Y 594.349,Z 229.447,A -85,B 0,C 180,E1 -1214.238,E2 -1214.238} C_VEL
LIN {X 0,Y 594.315,Z 229.452,A -85,B 0,C 180,E1 -1217.152,E2 -1217.152} C_VEL
LIN {X 0,Y 594.332,Z 229.447,A -85,B 0,C 180,E1 -1219.429,E2 -1219.429} C_VEL
LIN {X 0,Y 594.35,Z 229.454,A -85,B 0,C 180,E1 -1222.395,E2 -1222.395} C_VEL
LIN {X 0,Y 594.352,Z 229.445,A -85,B 0,C 180,E1 -1225.418,E2 -1225.418} C_VEL
LIN {X 0,Y 594.364,Z 229.45,A -85,B 0,C 180,E1 -1228.357,E2 -1228.357} C_VEL
LIN {X 0,Y 594.365,Z 229.443,A -85,B 0,C 180,E1 -1231.043,E2 -1231.043} C_VEL
LIN {X 0,Y 594.363,Z 229.451,A -85,B 0,C 180,E1 -1234.055,E2 -1234.055} C_VEL
LIN {X 0,Y 594.369,Z 229.446,A -85,B 0,C 180,E1 -1236.294,E2 -1236.294} C_VEL
LIN {X 0,Y 594.388,Z 229.443,A -85,B 0,C 180,E1 -1239.223,E2 -1239.223} C_VEL
LIN {X 0,Y 594.342,Z 229.448,A -85,B 0,C 180,E1 -1242.094,E2 -1242.094} C_VEL
LIN {X 0,Y 594.354,Z 229.445,A -85,B 0,C 180,E1 -1244.218,E2 -1244.218} C_VEL
LIN {X 0,Y 594.365,Z 229.443,A -85,B 0,C 180,E1 -1246.32,E2 -1246.32} C_VEL
LIN {X 0,Y 594.375,Z 229.449,A -85,B 0,C 180,E1 -1249.094,E2 -1249.094} C_VEL
LIN {X 0,Y 594.405,Z 229.439,A -85,B 0,C 180,E1 -1251.842,E2 -1251.842} C_VEL
LIN {X 0,Y 594.379,Z 229.445,A -85,B 0,C 180,E1 -1254.571,E2 -1254.571} C_VEL
LIN {X 0,Y 594.409,Z 229.442,A -85,B 0,C 180,E1 -1257.288,E2 -1257.288} C_VEL
LIN {X 0,Y 594.396,Z 229.44,A -85,B 0,C 180,E1 -1259.999,E2 -1259.999} C_VEL
LIN {X 0,Y 594.407,Z 229.447,A -85,B 0,C 180,E1 -1262.71,E2 -1262.71} C_VEL
LIN {X 0,Y 594.392,Z 229.44,A -85,B 0,C 180,E1 -1265.427,E2 -1265.427} C_VEL
LIN {X 0,Y 594.407,Z 229.443,A -85,B 0,C 180,E1 -1268.156,E2 -1268.156} C_VEL
LIN {X 0,Y 594.386,Z 229.441,A -85,B 0,C 180,E1 -1271.078,E2 -1271.078} C_VEL
LIN {X 0,Y 594.377,Z 229.444,A -85,B 0,C 180,E1 -1273.678,E2 -1273.678} C_VEL
LIN {X 0,Y 594.357,Z 229.445,A -85,B 0,C 180,E1 -1275.341,E2 -1275.341} C_VEL
LIN {X 0,Y 593.69,Z 229.535,A -85,B 0,C 180,E1 -1275.906,E2 -1275.906} C_VEL
LIN {X 0,Y 590.837,Z 229.893,A -85,B 0,C 180,E1 -1276.825,E2 -1276.825} C_VEL
LIN {X 0,Y 588.43,Z 230.194,A -85,B 0,C 180,E1 -1277.563,E2 -1277.563} C_VEL
LIN {X 0,Y 587.4,Z 230.319,A -85,B 0,C 180,E1 -1278.133,E2 -1278.133} C_VEL
LIN {X 0,Y 587.318,Z 230.326,A -85,B 0,C 180,E1 -1278.326,E2 -1278.326} C_VEL
LIN {X 0,Y 587.345,Z 230.318,A -85,B 0,C 180,E1 -1281.044,E2 -1281.044} C_VEL
LIN {X 0,Y 587.328,Z 230.326,A -85,B 0,C 180,E1 -1284.006,E2 -1284.006} C_VEL
LIN {X 0,Y 587.354,Z 230.318,A -85,B 0,C 180,E1 -1286.277,E2 -1286.277} C_VEL
LIN {X 0,Y 587.342,Z 230.322,A -85,B 0,C 180,E1 -1289.134,E2 -1289.134} C_VEL
LIN {X 0,Y 587.344,Z 230.321,A -85,B 0,C 180,E1 -1291.838,E2 -1291.838} C_VEL
LIN {X 0,Y 587.346,Z 230.317,A -85,B 0,C 180,E1 -1294.349,E2 -1294.349} C_VEL
LIN {X 0,Y 587.341,Z 230.321,A -85,B 0,C 180,E1 -1296.746,E2 -1296.746} C_VEL
LIN {X 0,Y 587.335,Z 230.324,A -85,B 0,C 180,E1 -1299.359,E2 -1299.359} C_VEL
LIN {X 0,Y 587.353,Z 230.317,A -85,B 0,C 180,E1 -1302.111,E2 -1302.111} C_VEL
LIN {X 0,Y 587.302,Z 230.329,A -85,B 0,C 180,E1 -1305.089,E2 -1305.089} C_VEL
LIN {X 0,Y 587.339,Z 230.318,A -85,B 0,C 180,E1 -1307.927,E2 -1307.927} C_VEL
LIN {X 0,Y 587.32,Z 230.324,A -85,B 0,C 180,E1 -1311.058,E2 -1311.058} C_VEL
LIN {X 0,Y 587.339,Z 230.319,A -85,B 0,C 180,E1 -1313.292,E2 -1313.292} C_VEL
LIN {X 0,Y 587.348,Z 230.319,A -85,B 0,C 180,E1 -1315.78,E2 -1315.78} C_VEL
LIN {X 0,Y 587.327,Z 230.329,A -85,B 0,C 180,E1 -1318.231,E2 -1318.231} C_VEL
LIN {X 0,Y 587.333,Z 230.32,A -85,B 0,C 180,E1 -1320.867,E2 -1320.867} C_VEL
LIN {X 0,Y 587.324,Z 230.327,A -85,B 0,C 180,E1 -1323.823,E2 -1323.823} C_VEL
LIN {X 0,Y 587.318,Z 230.33,A -85,B 0,C 180,E1 -1325.993,E2 -1325.993} C_VEL
LIN {X 0,Y 587.297,Z 230.327,A -85,B 0,C 180,E1 -1327.485,E2 -1327.485} C_VEL
LIN {X 0,Y 587.273,Z 231.085,A -85,B 0,C 180,E1 -1328.224,E2 -1328.224} C_VEL
LIN {X 0,Y 587.282,Z 236.052,A -85,B 0,C 180,E1 -1331.149,E2 -1331.149} C_VEL
LIN {X 0,Y 587.296,Z 239.768,A -85,B 0,C 180,E1 -1333.31,E2 -1333.31} C_VEL
LIN {X 0,Y 587.232,Z 244.771,A -85,B 0,C 180,E1 -1336.152,E2 -1336.152} C_VEL
LIN {X 0,Y 587.237,Z 249.752,A -85,B 0,C 180,E1 -1338.961,E2 -1338.961} C_VEL
LIN {X 0,Y 587.216,Z 254.929,A -85,B 0,C 180,E1 -1341.743,E2 -1341.743} C_VEL
LIN {X 0,Y 587.192,Z 258.852,A -85,B 0,C 180,E1 -1343.816,E2 -1343.816} C_VEL
LIN {X 0,Y 587.164,Z 262.81,A -85,B 0,C 180,E1 -1345.882,E2 -1345.882} C_VEL
LIN {X 0,Y 587.146,Z 268.139,A -85,B 0,C 180,E1 -1348.628,E2 -1348.628} C_VEL
LIN {X 0,Y 587.17,Z 272.554,A -85,B 0,C 180,E1 -1350.879,E2 -1350.879} C_VEL
LIN {X 0,Y 587.735,Z 278.373,A -85,B 0,C 180,E1 -1351.006,E2 -1351.006} C_VEL
LIN {X 0,Y 587.626,Z 291.559,A -85,B 0,C 180,E1 -1351.371,E2 -1351.371} C_VEL
LIN {X 0,Y 587.515,Z 302.654,A -85,B 0,C 180,E1 -1351.799,E2 -1351.799} C_VEL
LIN {X 0,Y 587.511,Z 314.496,A -85,B 0,C 180,E1 -1352.399,E2 -1352.399} C_VEL
LIN {X 0,Y 587.449,Z 325.169,A -85,B 0,C 180,E1 -1353.086,E2 -1353.086} C_VEL
LIN {X 0,Y 587.366,Z 335.848,A -85,B 0,C 180,E1 -1353.945,E2 -1353.945} C_VEL
LIN {X 0,Y 587.295,Z 344.566,A -85,B 0,C 180,E1 -1354.805,E2 -1354.805} C_VEL
LIN {X 0,Y 587.252,Z 353.087,A -85,B 0,C 180,E1 -1355.838,E2 -1355.838} C_VEL
LIN {X 0,Y 587.215,Z 359.939,A -85,B 0,C 180,E1 -1356.874,E2 -1356.874} C_VEL
LIN {X 0,Y 587.198,Z 365.441,A -85,B 0,C 180,E1 -1357.911,E2 -1357.911} C_VEL
LIN {X 0,Y 587.152,Z 369.768,A -85,B 0,C 180,E1 -1358.952,E2 -1358.952} C_VEL
LIN {X 0,Y 587.156,Z 372.058,A -85,B 0,C 180,E1 -1359.647,E2 -1359.647} C_VEL
LIN {X 0,Y 587.14,Z 373.908,A -85,B 0,C 180,E1 -1360.343,E2 -1360.343} C_VEL
LIN {X 0,Y 587.184,Z 375.316,A -85,B 0,C 180,E1 -1361.058,E2 -1361.058} C_VEL
LIN {X 0,Y 587.155,Z 376.84,A -85,B 0,C 180,E1 -1362.442,E2 -1362.442} C_VEL
LIN {X 0,Y 587.14,Z 376.983,A -85,B 0,C 180,E1 -1363.145,E2 -1363.145} C_VEL
LIN {X 0,Y 587.146,Z 376.453,A -85,B 0,C 180,E1 -1364.181,E2 -1364.181} C_VEL
LIN {X 0,Y 587.139,Z 374.912,A -85,B 0,C 180,E1 -1365.268,E2 -1365.268} C_VEL
LIN {X 0,Y 587.153,Z 372.384,A -85,B 0,C 180,E1 -1366.337,E2 -1366.337} C_VEL
LIN {X 0,Y 587.167,Z 368.767,A -85,B 0,C 180,E1 -1367.411,E2 -1367.411} C_VEL
LIN {X 0,Y 587.214,Z 363.934,A -85,B 0,C 180,E1 -1368.491,E2 -1368.491} C_VEL
LIN {X 0,Y 587.24,Z 357.709,A -85,B 0,C 180,E1 -1369.578,E2 -1369.578} C_VEL
LIN {X 0,Y 587.279,Z 349.839,A -85,B 0,C 180,E1 -1370.672,E2 -1370.672} C_VEL
LIN {X 0,Y 587.309,Z 341.696,A -85,B 0,C 180,E1 -1371.59,E2 -1371.59} C_VEL
LIN {X 0,Y 587.41,Z 331.58,A -85,B 0,C 180,E1 -1372.51,E2 -1372.51} C_VEL
LIN {X 0,Y 587.414,Z 321.54,A -85,B 0,C 180,E1 -1373.254,E2 -1373.254} C_VEL
LIN {X 0,Y 587.455,Z 310.611,A -85,B 0,C 180,E1 -1373.907,E2 -1373.907} C_VEL
LIN {X 0,Y 587.581,Z 298.22,A -85,B 0,C 180,E1 -1374.477,E2 -1374.477} C_VEL
LIN {X 0,Y 587.678,Z 285.389,A -85,B 0,C 180,E1 -1374.908,E2 -1374.908} C_VEL
LIN {X 0,Y 587.505,Z 275.135,A -85,B 0,C 180,E1 -1375.153,E2 -1375.153} C_VEL
LIN {X 0,Y 587.146,Z 272.545,A -85,B 0,C 180,E1 -1375.216,E2 -1375.216} C_VEL
LIN {X 0,Y 587.127,Z 267.425,A -85,B 0,C 180,E1 -1377.828,E2 -1377.828} C_VEL
LIN {X 0,Y 587.152,Z 262.285,A -85,B 0,C 180,E1 -1380.482,E2 -1380.482} C_VEL
LIN {X 0,Y 587.147,Z 257.314,A -85,B 0,C 180,E1 -1383.085,E2 -1383.085} C_VEL
LIN {X 0,Y 587.186,Z 252.018,A -85,B 0,C 180,E1 -1385.906,E2 -1385.906} C_VEL
LIN {X 0,Y 587.21,Z 246.548,A -85,B 0,C 180,E1 -1388.929,E2 -1388.929} C_VEL
LIN {X 0,Y 587.234,Z 241.009,A -85,B 0,C 180,E1 -1392.099,E2 -1392.099} C_VEL
LIN {X 0,Y 587.261,Z 235.808,A -85,B 0,C 180,E1 -1395.085,E2 -1395.085} C_VEL
LIN {X 0,Y 587.292,Z 231.019,A -85,B 0,C 180,E1 -1397.924,E2 -1397.924} C_VEL
LIN {X 0,Y 587.318,Z 230.326,A -85,B 0,C 180,E1 -1398.925,E2 -1398.925} C_VEL
LIN {X 0,Y 587.316,Z 230.328,A -85,B 0,C 180,E1 -1401.521,E2 -1401.521} C_VEL
LIN {X 0,Y 587.34,Z 230.326,A -85,B 0,C 180,E1 -1404.455,E2 -1404.455} C_VEL
LIN {X 0,Y 587.321,Z 230.326,A -85,B 0,C 180,E1 -1406.889,E2 -1406.889} C_VEL
LIN {X 0,Y 587.339,Z 230.322,A -85,B 0,C 180,E1 -1409.487,E2 -1409.487} C_VEL
LIN {X 0,Y 587.338,Z 230.323,A -85,B 0,C 180,E1 -1412.307,E2 -1412.307} C_VEL
LIN {X 0,Y 587.339,Z 230.322,A -85,B 0,C 180,E1 -1415.42,E2 -1415.42} C_VEL
LIN {X 0,Y 587.357,Z 230.321,A -85,B 0,C 180,E1 -1417.488,E2 -1417.488} C_VEL
LIN {X 0,Y 587.318,Z 230.327,A -85,B 0,C 180,E1 -1419.696,E2 -1419.696} C_VEL
LIN {X 0,Y 587.346,Z 230.324,A -85,B 0,C 180,E1 -1422.595,E2 -1422.595} C_VEL
LIN {X 0,Y 587.343,Z 230.323,A -85,B 0,C 180,E1 -1425.743,E2 -1425.743} C_VEL
LIN {X 0,Y 587.334,Z 230.324,A -85,B 0,C 180,E1 -1428.867,E2 -1428.867} C_VEL
LIN {X 0,Y 587.36,Z 230.322,A -85,B 0,C 180,E1 -1431.746,E2 -1431.746} C_VEL
LIN {X 0,Y 587.348,Z 230.326,A -85,B 0,C 180,E1 -1434.508,E2 -1434.508} C_VEL
LIN {X 0,Y 587.376,Z 230.321,A -85,B 0,C 180,E1 -1437.258,E2 -1437.258} C_VEL
LIN {X 0,Y 587.358,Z 230.32,A -85,B 0,C 180,E1 -1440.001,E2 -1440.001} C_VEL
LIN {X 0,Y 587.37,Z 230.318,A -85,B 0,C 180,E1 -1442.744,E2 -1442.744} C_VEL
LIN {X 0,Y 587.345,Z 230.322,A -85,B 0,C 180,E1 -1445.494,E2 -1445.494} C_VEL
LIN {X 0,Y 587.356,Z 230.323,A -85,B 0,C 180,E1 -1448.256,E2 -1448.256} C_VEL
LIN {X 0,Y 587.353,Z 230.325,A -85,B 0,C 180,E1 -1451.142,E2 -1451.142} C_VEL
LIN {X 0,Y 587.33,Z 230.327,A -85,B 0,C 180,E1 -1454.252,E2 -1454.252} C_VEL
LIN {X 0,Y 587.354,Z 230.323,A -85,B 0,C 180,E1 -1457.407,E2 -1457.407} C_VEL
LIN {X 0,Y 587.313,Z 230.329,A -85,B 0,C 180,E1 -1460.306,E2 -1460.306} C_VEL
LIN {X 0,Y 587.318,Z 230.33,A -85,B 0,C 180,E1 -1463.26,E2 -1463.26} C_VEL
LIN {X 0,Y 587.33,Z 230.324,A -85,B 0,C 180,E1 -1465.517,E2 -1465.517} C_VEL
LIN {X 0,Y 587.296,Z 230.332,A -85,B 0,C 180,E1 -1467.821,E2 -1467.821} C_VEL
LIN {X 0,Y 587.336,Z 230.327,A -85,B 0,C 180,E1 -1470.512,E2 -1470.512} C_VEL
LIN {X 0,Y 587.332,Z 230.323,A -85,B 0,C 180,E1 -1473.113,E2 -1473.113} C_VEL
LIN {X 0,Y 587.29,Z 230.33,A -85,B 0,C 180,E1 -1475.539,E2 -1475.539} C_VEL
LIN {X 0,Y 587.339,Z 230.324,A -85,B 0,C 180,E1 -1477.84,E2 -1477.84} C_VEL
LIN {X 0,Y 587.308,Z 230.326,A -85,B 0,C 180,E1 -1480.255,E2 -1480.255} C_VEL
LIN {X 0,Y 587.32,Z 230.326,A -85,B 0,C 180,E1 -1483.12,E2 -1483.12} C_VEL
LIN {X 0,Y 587.306,Z 230.329,A -85,B 0,C 180,E1 -1486.049,E2 -1486.049} C_VEL
LIN {X 0,Y 587.332,Z 230.328,A -85,B 0,C 180,E1 -1488.926,E2 -1488.926} C_VEL
LIN {X 0,Y 587.334,Z 230.326,A -85,B 0,C 180,E1 -1491.522,E2 -1491.522} C_VEL
LIN {X 0,Y 587.342,Z 230.41,A -85,B 0,C 180,E1 -1493.999,E2 -1493.999} C_VEL
LIN {X 0,Y 587.514,Z 234.62,A -85,B 0,C 180,E1 -1495.629,E2 -1495.629} C_VEL
LIN {X 0,Y 587.458,Z 241.69,A -85,B 0,C 180,E1 -1498.239,E2 -1498.239} C_VEL
LIN {X 0,Y 587.392,Z 248.994,A -85,B 0,C 180,E1 -1500.86,E2 -1500.86} C_VEL
LIN {X 0,Y 587.364,Z 257.682,A -85,B 0,C 180,E1 -1503.819,E2 -1503.819} C_VEL
LIN {X 0,Y 587.33,Z 266.337,A -85,B 0,C 180,E1 -1506.742,E2 -1506.742} C_VEL
LIN {X 0,Y 587.294,Z 274.143,A -85,B 0,C 180,E1 -1509.334,E2 -1509.334} C_VEL
LIN {X 0,Y 587.281,Z 283.032,A -85,B 0,C 180,E1 -1512.233,E2 -1512.233} C_VEL
LIN {X 0,Y 587.218,Z 291.936,A -85,B 0,C 180,E1 -1515.089,E2 -1515.089} C_VEL
LIN {X 0,Y 587.173,Z 300.493,A -85,B 0,C 180,E1 -1517.8,E2 -1517.8} C_VEL
LIN {X 0,Y 587.747,Z 305.247,A -85,B 0,C 180,E1 -1517.9,E2 -1517.9} C_VEL
LIN {X 0,Y 587.679,Z 318.508,A -85,B 0,C 180,E1 -1518.227,E2 -1518.227} C_VEL
LIN {X 0,Y 587.566,Z 330.467,A -85,B 0,C 180,E1 -1518.659,E2 -1518.659} C_VEL
LIN {X 0,Y 587.49,Z 342.217,A -85,B 0,C 180,E1 -1519.227,E2 -1519.227} C_VEL
LIN {X 0,Y 587.457,Z 353.483,A -85,B 0,C 180,E1 -1519.924,E2 -1519.924} C_VEL
LIN {X 0,Y 587.384,Z 363.65,A -85,B 0,C 180,E1 -1520.705,E2 -1520.705} C_VEL
LIN {X 0,Y 587.34,Z 372.789,A -85,B 0,C 180,E1 -1521.571,E2 -1521.571} C_VEL
LIN {X 0,Y 587.259,Z 381.692,A -85,B 0,C 180,E1 -1522.609,E2 -1522.609} C_VEL
LIN {X 0,Y 587.195,Z 388.748,A -85,B 0,C 180,E1 -1523.628,E2 -1523.628} C_VEL
LIN {X 0,Y 587.211,Z 393.681,A -85,B 0,C 180,E1 -1524.506,E2 -1524.506} C_VEL
LIN {X 0,Y 587.188,Z 398.372,A -85,B 0,C 180,E1 -1525.538,E2 -1525.538} C_VEL
LIN {X 0,Y 587.193,Z 401.957,A -85,B 0,C 180,E1 -1526.569,E2 -1526.569} C_VEL
LIN {X 0,Y 587.132,Z 403.809,A -85,B 0,C 180,E1 -1527.256,E2 -1527.256} C_VEL
LIN {X 0,Y 587.141,Z 405.2,A -85,B 0,C 180,E1 -1527.942,E2 -1527.942} C_VEL
LIN {X 0,Y 587.14,Z 406.784,A -85,B 0,C 180,E1 -1529.314,E2 -1529.314} C_VEL
LIN {X 0,Y 587.137,Z 407,A -85,B 0,C 180,E1 -1530,E2 -1530} C_VEL
LIN {X 0,Y 587.147,Z 406.185,A -85,B 0,C 180,E1 -1531.372,E2 -1531.372} C_VEL
LIN {X 0,Y 587.141,Z 405.201,A -85,B 0,C 180,E1 -1532.058,E2 -1532.058} C_VEL
LIN {X 0,Y 587.132,Z 403.81,A -85,B 0,C 180,E1 -1532.744,E2 -1532.744} C_VEL
LIN {X 0,Y 587.213,Z 400.896,A -85,B 0,C 180,E1 -1533.774,E2 -1533.774} C_VEL
LIN {X 0,Y 587.147,Z 396.95,A -85,B 0,C 180,E1 -1534.806,E2 -1534.806} C_VEL
LIN {X 0,Y 587.218,Z 390.878,A -85,B 0,C 180,E1 -1536.011,E2 -1536.011} C_VEL
LIN {X 0,Y 587.245,Z 384.238,A -85,B 0,C 180,E1 -1537.046,E2 -1537.046} C_VEL
LIN {X 0,Y 587.299,Z 375.991,A -85,B 0,C 180,E1 -1538.083,E2 -1538.083} C_VEL
LIN {X 0,Y 587.343,Z 367.54,A -85,B 0,C 180,E1 -1538.949,E2 -1538.949} C_VEL
LIN {X 0,Y 587.415,Z 357.098,A -85,B 0,C 180,E1 -1539.816,E2 -1539.816} C_VEL
LIN {X 0,Y 587.451,Z 346.761,A -85,B 0,C 180,E1 -1540.512,E2 -1540.512} C_VEL
LIN {X 0,Y 587.529,Z 335.174,A -85,B 0,C 180,E1 -1541.133,E2 -1541.133} C_VEL
LIN {X 0,Y 587.607,Z 322.705,A -85,B 0,C 180,E1 -1541.636,E2 -1541.636} C_VEL
LIN {X 0,Y 587.744,Z 309.446,A -85,B 0,C 180,E1 -1542.013,E2 -1542.013} C_VEL
LIN {X 0,Y 587.528,Z 302.664,A -85,B 0,C 180,E1 -1542.154,E2 -1542.154} C_VEL
LIN {X 0,Y 587.173,Z 300.423,A -85,B 0,C 180,E1 -1542.222,E2 -1542.222} C_VEL
LIN {X 0,Y 587.219,Z 291.936,A -85,B 0,C 180,E1 -1544.911,E2 -1544.911} C_VEL
LIN {X 0,Y 587.281,Z 283.032,A -85,B 0,C 180,E1 -1547.767,E2 -1547.767} C_VEL
LIN {X 0,Y 587.294,Z 274.143,A -85,B 0,C 180,E1 -1550.667,E2 -1550.667} C_VEL
LIN {X 0,Y 587.346,Z 265.223,A -85,B 0,C 180,E1 -1553.631,E2 -1553.631} C_VEL
LIN {X 0,Y 587.364,Z 257.371,A -85,B 0,C 180,E1 -1556.277,E2 -1556.277} C_VEL
LIN {X 0,Y 587.367,Z 249.043,A -85,B 0,C 180,E1 -1559.136,E2 -1559.136} C_VEL
LIN {X 0,Y 587.459,Z 241.441,A -85,B 0,C 180,E1 -1561.853,E2 -1561.853} C_VEL
LIN {X 0,Y 587.531,Z 234.627,A -85,B 0,C 180,E1 -1564.373,E2 -1564.373} C_VEL
LIN {X 0,Y 587.303,Z 230.33,A -85,B 0,C 180,E1 -1566.057,E2 -1566.057} C_VEL
LIN {X 0,Y 587.307,Z 230.326,A -85,B 0,C 180,E1 -1568.48,E2 -1568.48} C_VEL
LIN {X 0,Y 587.296,Z 230.33,A -85,B 0,C 180,E1 -1571.159,E2 -1571.159} C_VEL
LIN {X 0,Y 587.296,Z 230.325,A -85,B 0,C 180,E1 -1574.11,E2 -1574.11} C_VEL
LIN {X 0,Y 587.273,Z 230.331,A -85,B 0,C 180,E1 -1576.989,E2 -1576.989} C_VEL
LIN {X 0,Y 587.285,Z 230.326,A -85,B 0,C 180,E1 -1579.743,E2 -1579.743} C_VEL
LIN {X 0,Y 587.305,Z 230.332,A -85,B 0,C 180,E1 -1582.389,E2 -1582.389} C_VEL
LIN {X 0,Y 587.326,Z 230.321,A -85,B 0,C 180,E1 -1585.654,E2 -1585.654} C_VEL
LIN {X 0,Y 587.324,Z 230.329,A -85,B 0,C 180,E1 -1588.229,E2 -1588.229} C_VEL
LIN {X 0,Y 587.335,Z 230.319,A -85,B 0,C 180,E1 -1590.867,E2 -1590.867} C_VEL
LIN {X 0,Y 587.301,Z 230.331,A -85,B 0,C 180,E1 -1593.828,E2 -1593.828} C_VEL
LIN {X 0,Y 587.322,Z 230.328,A -85,B 0,C 180,E1 -1595.992,E2 -1595.992} C_VEL
LIN {X 0,Y 587.309,Z 230.325,A -85,B 0,C 180,E1 -1598.225,E2 -1598.225} C_VEL
LIN {X 0,Y 587.337,Z 230.322,A -85,B 0,C 180,E1 -1601.15,E2 -1601.15} C_VEL
LIN {X 0,Y 587.314,Z 230.324,A -85,B 0,C 180,E1 -1604.024,E2 -1604.024} C_VEL
LIN {X 0,Y 587.345,Z 230.318,A -85,B 0,C 180,E1 -1606.153,E2 -1606.153} C_VEL
LIN {X 0,Y 587.339,Z 230.323,A -85,B 0,C 180,E1 -1608.962,E2 -1608.962} C_VEL
LIN {X 0,Y 587.36,Z 230.318,A -85,B 0,C 180,E1 -1611.744,E2 -1611.744} C_VEL
LIN {X 0,Y 587.344,Z 230.32,A -85,B 0,C 180,E1 -1614.506,E2 -1614.506} C_VEL
LIN {X 0,Y 587.374,Z 230.319,A -85,B 0,C 180,E1 -1617.256,E2 -1617.256} C_VEL
LIN {X 0,Y 587.366,Z 230.316,A -85,B 0,C 180,E1 -1619.999,E2 -1619.999} C_VEL
LIN {X 0,Y 587.372,Z 230.323,A -85,B 0,C 180,E1 -1622.742,E2 -1622.742} C_VEL
LIN {X 0,Y 587.355,Z 230.317,A -85,B 0,C 180,E1 -1625.492,E2 -1625.492} C_VEL
LIN {X 0,Y 587.361,Z 230.323,A -85,B 0,C 180,E1 -1628.254,E2 -1628.254} C_VEL
LIN {X 0,Y 587.351,Z 230.317,A -85,B 0,C 180,E1 -1631.141,E2 -1631.141} C_VEL
LIN {X 0,Y 587.353,Z 230.325,A -85,B 0,C 180,E1 -1634.26,E2 -1634.26} C_VEL
LIN {X 0,Y 587.35,Z 230.318,A -85,B 0,C 180,E1 -1637.405,E2 -1637.405} C_VEL
LIN {X 0,Y 587.318,Z 230.326,A -85,B 0,C 180,E1 -1638.326,E2 -1638.326} C_VEL
LIN {X 0,Y 586.663,Z 230.405,A -85,B 0,C 180,E1 -1638.898,E2 -1638.898} C_VEL
LIN {X 0,Y 583.831,Z 230.764,A -85,B 0,C 180,E1 -1639.827,E2 -1639.827} C_VEL
LIN {X 0,Y 581.421,Z 231.061,A -85,B 0,C 180,E1 -1640.574,E2 -1640.574} C_VEL
LIN {X 0,Y 580.369,Z 231.189,A -85,B 0,C 180,E1 -1641.15,E2 -1641.15} C_VEL
LIN {X 0,Y 580.275,Z 231.2,A -85,B 0,C 180,E1 -1641.345,E2 -1641.345} C_VEL
LIN {X 0,Y 580.29,Z 231.199,A -85,B 0,C 180,E1 -1644.316,E2 -1644.316} C_VEL
LIN {X 0,Y 580.3,Z 231.195,A -85,B 0,C 180,E1 -1646.621,E2 -1646.621} C_VEL
LIN {X 0,Y 580.296,Z 231.202,A -85,B 0,C 180,E1 -1649.311,E2 -1649.311} C_VEL
LIN {X 0,Y 580.291,Z 231.197,A -85,B 0,C 180,E1 -1652.2,E2 -1652.2} C_VEL
LIN {X 0,Y 580.29,Z 231.198,A -85,B 0,C 180,E1 -1654.695,E2 -1654.695} C_VEL
LIN {X 0,Y 580.288,Z 231.205,A -85,B 0,C 180,E1 -1657.268,E2 -1657.268} C_VEL
LIN {X 0,Y 580.294,Z 231.196,A -85,B 0,C 180,E1 -1660.272,E2 -1660.272} C_VEL
LIN {X 0,Y 580.285,Z 231.203,A -85,B 0,C 180,E1 -1662.704,E2 -1662.704} C_VEL
LIN {X 0,Y 580.26,Z 231.2,A -85,B 0,C 180,E1 -1665.608,E2 -1665.608} C_VEL
LIN {X 0,Y 580.301,Z 231.198,A -85,B 0,C 180,E1 -1668.234,E2 -1668.234} C_VEL
LIN {X 0,Y 580.275,Z 231.202,A -85,B 0,C 180,E1 -1670.966,E2 -1670.966} C_VEL
LIN {X 0,Y 580.267,Z 231.199,A -85,B 0,C 180,E1 -1673.597,E2 -1673.597} C_VEL
LIN {X 0,Y 580.304,Z 231.201,A -85,B 0,C 180,E1 -1676.145,E2 -1676.145} C_VEL
LIN {X 0,Y 580.263,Z 231.204,A -85,B 0,C 180,E1 -1678.615,E2 -1678.615} C_VEL
LIN {X 0,Y 580.277,Z 231.198,A -85,B 0,C 180,E1 -1681.024,E2 -1681.024} C_VEL
LIN {X 0,Y 580.272,Z 231.203,A -85,B 0,C 180,E1 -1683.667,E2 -1683.667} C_VEL
LIN {X 0,Y 580.285,Z 231.202,A -85,B 0,C 180,E1 -1685.684,E2 -1685.684} C_VEL
LIN {X 0,Y 580.271,Z 231.2,A -85,B 0,C 180,E1 -1687.197,E2 -1687.197} C_VEL
LIN {X 0,Y 580.222,Z 231.458,A -85,B 0,C 180,E1 -1687.946,E2 -1687.946} C_VEL
LIN {X 0,Y 580.25,Z 236.423,A -85,B 0,C 180,E1 -1690.912,E2 -1690.912} C_VEL
LIN {X 0,Y 580.208,Z 241.39,A -85,B 0,C 180,E1 -1693.824,E2 -1693.824} C_VEL
LIN {X 0,Y 580.152,Z 246.407,A -85,B 0,C 180,E1 -1696.693,E2 -1696.693} C_VEL
LIN {X 0,Y 580.148,Z 251.388,A -85,B 0,C 180,E1 -1699.531,E2 -1699.531} C_VEL
LIN {X 0,Y 580.138,Z 256.55,A -85,B 0,C 180,E1 -1702.342,E2 -1702.342} C_VEL
LIN {X 0,Y 580.153,Z 261.8,A -85,B 0,C 180,E1 -1705.136,E2 -1705.136} C_VEL
LIN {X 0,Y 580.051,Z 267.117,A -85,B 0,C 180,E1 -1707.917,E2 -1707.917} C_VEL
LIN {X 0,Y 580.07,Z 271.14,A -85,B 0,C 180,E1 -1710,E2 -1710} C_VEL
LIN {X 0,Y 580.072,Z 272.531,A -85,B 0,C 180,E1 -1710.716,E2 -1710.716} C_VEL
LIN {X 0,Y 580.798,Z 278.635,A -85,B 0,C 180,E1 -1710.867,E2 -1710.867} C_VEL
LIN {X 0,Y 580.686,Z 291.103,A -85,B 0,C 180,E1 -1711.214,E2 -1711.214} C_VEL
LIN {X 0,Y 580.535,Z 302.325,A -85,B 0,C 180,E1 -1711.648,E2 -1711.648} C_VEL
LIN {X 0,Y 580.501,Z 314.241,A -85,B 0,C 180,E1 -1712.255,E2 -1712.255} C_VEL
LIN {X 0,Y 580.427,Z 324.973,A -85,B 0,C 180,E1 -1712.95,E2 -1712.95} C_VEL
LIN {X 0,Y 580.328,Z 335.687,A -85,B 0,C 180,E1 -1713.819,E2 -1713.819} C_VEL
LIN {X 0,Y 580.251,Z 344.428,A -85,B 0,C 180,E1 -1714.689,E2 -1714.689} C_VEL
LIN {X 0,Y 580.173,Z 352.985,A -85,B 0,C 180,E1 -1715.735,E2 -1715.735} C_VEL
LIN {X 0,Y 580.172,Z 359.014,A -85,B 0,C 180,E1 -1716.639,E2 -1716.639} C_VEL
LIN {X 0,Y 580.11,Z 364.561,A -85,B 0,C 180,E1 -1717.658,E2 -1717.658} C_VEL
LIN {X 0,Y 580.084,Z 369.086,A -85,B 0,C 180,E1 -1718.71,E2 -1718.71} C_VEL
LIN {X 0,Y 580.061,Z 372.531,A -85,B 0,C 180,E1 -1719.766,E2 -1719.766} C_VEL
LIN {X 0,Y 580.098,Z 375.415,A -85,B 0,C 180,E1 -1721.096,E2 -1721.096} C_VEL
LIN {X 0,Y 580.046,Z 376.444,A -85,B 0,C 180,E1 -1721.886,E2 -1721.886} C_VEL
LIN {X 0,Y 580.045,Z 376.905,A -85,B 0,C 180,E1 -1722.597,E2 -1722.597} C_VEL
LIN {X 0,Y 580.053,Z 376.947,A -85,B 0,C 180,E1 -1723.309,E2 -1723.309} C_VEL
LIN {X 0,Y 580.053,Z 376.4,A -85,B 0,C 180,E1 -1724.242,E2 -1724.242} C_VEL
LIN {X 0,Y 580.056,Z 374.575,A -85,B 0,C 180,E1 -1725.459,E2 -1725.459} C_VEL
LIN {X 0,Y 580.066,Z 372.901,A -85,B 0,C 180,E1 -1726.18,E2 -1726.18} C_VEL
LIN {X 0,Y 580.067,Z 369.487,A -85,B 0,C 180,E1 -1727.267,E2 -1727.267} C_VEL
LIN {X 0,Y 580.102,Z 364.895,A -85,B 0,C 180,E1 -1728.36,E2 -1728.36} C_VEL
LIN {X 0,Y 580.175,Z 359.189,A -85,B 0,C 180,E1 -1729.421,E2 -1729.421} C_VEL
LIN {X 0,Y 580.181,Z 351.393,A -85,B 0,C 180,E1 -1730.566,E2 -1730.566} C_VEL
LIN {X 0,Y 580.244,Z 343.575,A -85,B 0,C 180,E1 -1731.493,E2 -1731.493} C_VEL
LIN {X 0,Y 580.346,Z 333.989,A -85,B 0,C 180,E1 -1732.424,E2 -1732.424} C_VEL
LIN {X 0,Y 580.397,Z 323.357,A -85,B 0,C 180,E1 -1733.254,E2 -1733.254} C_VEL
LIN {X 0,Y 580.461,Z 312.597,A -85,B 0,C 180,E1 -1733.928,E2 -1733.928} C_VEL
LIN {X 0,Y 580.575,Z 300.695,A -85,B 0,C 180,E1 -1734.514,E2 -1734.514} C_VEL
LIN {X 0,Y 580.726,Z 288.111,A -85,B 0,C 180,E1 -1734.973,E2 -1734.973} C_VEL
LIN {X 0,Y 580.628,Z 276.252,A -85,B 0,C 180,E1 -1735.276,E2 -1735.276} C_VEL
LIN {X 0,Y 580.054,Z 272.524,A -85,B 0,C 180,E1 -1735.379,E2 -1735.379} C_VEL
LIN {X 0,Y 580.048,Z 267.069,A -85,B 0,C 180,E1 -1738.198,E2 -1738.198} C_VEL
LIN {X 0,Y 580.059,Z 262.365,A -85,B 0,C 180,E1 -1740.66,E2 -1740.66} C_VEL
LIN {X 0,Y 580.077,Z 257.418,A -85,B 0,C 180,E1 -1743.285,E2 -1743.285} C_VEL
LIN {X 0,Y 580.117,Z 251.652,A -85,B 0,C 180,E1 -1746.414,E2 -1746.414} C_VEL
LIN {X 0,Y 580.138,Z 246.83,A -85,B 0,C 180,E1 -1749.168,E2 -1749.168} C_VEL
LIN {X 0,Y 580.17,Z 242.302,A -85,B 0,C 180,E1 -1751.777,E2 -1751.777} C_VEL
LIN {X 0,Y 580.216,Z 237.388,A -85,B 0,C 180,E1 -1754.63,E2 -1754.63} C_VEL
LIN {X 0,Y 580.254,Z 232.357,A -85,B 0,C 180,E1 -1757.63,E2 -1757.63} C_VEL
LIN {X 0,Y 580.23,Z 231.371,A -85,B 0,C 180,E1 -1758.228,E2 -1758.228} C_VEL
LIN {X 0,Y 580.271,Z 231.206,A -85,B 0,C 180,E1 -1760.067,E2 -1760.067} C_VEL
LIN {X 0,Y 580.29,Z 231.203,A -85,B 0,C 180,E1 -1763.065,E2 -1763.065} C_VEL
LIN {X 0,Y 580.287,Z 231.203,A -85,B 0,C 180,E1 -1765.441,E2 -1765.441} C_VEL
LIN {X 0,Y 580.294,Z 231.2,A -85,B 0,C 180,E1 -1767.968,E2 -1767.968} C_VEL
LIN {X 0,Y 580.298,Z 231.201,A -85,B 0,C 180,E1 -1770.689,E2 -1770.689} C_VEL
LIN {X 0,Y 580.259,Z 231.209,A -85,B 0,C 180,E1 -1773.377,E2 -1773.377} C_VEL
LIN {X 0,Y 580.288,Z 231.201,A -85,B 0,C 180,E1 -1775.684,E2 -1775.684} C_VEL
LIN {X 0,Y 580.277,Z 231.207,A -85,B 0,C 180,E1 -1777.949,E2 -1777.949} C_VEL
LIN {X 0,Y 580.284,Z 231.206,A -85,B 0,C 180,E1 -1780.914,E2 -1780.914} C_VEL
LIN {X 0,Y 580.275,Z 231.207,A -85,B 0,C 180,E1 -1783.826,E2 -1783.826} C_VEL
LIN {X 0,Y 580.304,Z 231.198,A -85,B 0,C 180,E1 -1785.984,E2 -1785.984} C_VEL
LIN {X 0,Y 580.291,Z 231.201,A -85,B 0,C 180,E1 -1788.828,E2 -1788.828} C_VEL
LIN {X 0,Y 580.325,Z 231.199,A -85,B 0,C 180,E1 -1791.645,E2 -1791.645} C_VEL
LIN {X 0,Y 580.311,Z 231.203,A -85,B 0,C 180,E1 -1794.441,E2 -1794.441} C_VEL
LIN {X 0,Y 580.341,Z 231.197,A -85,B 0,C 180,E1 -1797.224,E2 -1797.224} C_VEL
LIN {X 0,Y 580.328,Z 231.196,A -85,B 0,C 180,E1 -1800.001,E2 -1800.001} C_VEL
LIN {X 0,Y 580.336,Z 231.194,A -85,B 0,C 180,E1 -1802.777,E2 -1802.777} C_VEL
LIN {X 0,Y 580.311,Z 231.198,A -85,B 0,C 180,E1 -1805.561,E2 -1805.561} C_VEL
LIN {X 0,Y 580.319,Z 231.199,A -85,B 0,C 180,E1 -1808.357,E2 -1808.357} C_VEL
LIN {X 0,Y 580.324,Z 231.2,A -85,B 0,C 180,E1 -1811.209,E2 -1811.209} C_VEL
LIN {X 0,Y 580.302,Z 231.204,A -85,B 0,C 180,E1 -1814.018,E2 -1814.018} C_VEL
LIN {X 0,Y 580.303,Z 231.202,A -85,B 0,C 180,E1 -1816.915,E2 -1816.915} C_VEL
LIN {X 0,Y 580.277,Z 231.205,A -85,B 0,C 180,E1 -1819.824,E2 -1819.824} C_VEL
LIN {X 0,Y 580.261,Z 231.205,A -85,B 0,C 180,E1 -1822.054,E2 -1822.054} C_VEL
LIN {X 0,Y 580.301,Z 231.201,A -85,B 0,C 180,E1 -1825.081,E2 -1825.081} C_VEL
LIN {X 0,Y 580.271,Z 231.204,A -85,B 0,C 180,E1 -1828.188,E2 -1828.188} C_VEL
LIN {X 0,Y 580.287,Z 231.207,A -85,B 0,C 180,E1 -1830.697,E2 -1830.697} C_VEL
LIN {X 0,Y 580.297,Z 231.201,A -85,B 0,C 180,E1 -1833.317,E2 -1833.317} C_VEL
LIN {X 0,Y 580.24,Z 231.207,A -85,B 0,C 180,E1 -1835.757,E2 -1835.757} C_VEL
LIN {X 0,Y 580.285,Z 231.206,A -85,B 0,C 180,E1 -1838.147,E2 -1838.147} C_VEL
LIN {X 0,Y 580.291,Z 231.201,A -85,B 0,C 180,E1 -1840.845,E2 -1840.845} C_VEL
LIN {X 0,Y 580.284,Z 231.201,A -85,B 0,C 180,E1 -1843.658,E2 -1843.658} C_VEL
LIN {X 0,Y 580.236,Z 231.208,A -85,B 0,C 180,E1 -1846.614,E2 -1846.614} C_VEL
LIN {X 0,Y 580.293,Z 231.201,A -85,B 0,C 180,E1 -1849.73,E2 -1849.73} C_VEL
LIN {X 0,Y 580.298,Z 231.202,A -85,B 0,C 180,E1 -1852.733,E2 -1852.733} C_VEL
LIN {X 0,Y 580.277,Z 231.341,A -85,B 0,C 180,E1 -1853.854,E2 -1853.854} C_VEL
LIN {X 0,Y 580.527,Z 235.041,A -85,B 0,C 180,E1 -1855.321,E2 -1855.321} C_VEL
LIN {X 0,Y 580.45,Z 241.967,A -85,B 0,C 180,E1 -1857.947,E2 -1857.947} C_VEL
LIN {X 0,Y 580.381,Z 249.52,A -85,B 0,C 180,E1 -1860.677,E2 -1860.677} C_VEL
LIN {X 0,Y 580.319,Z 257.287,A -85,B 0,C 180,E1 -1863.379,E2 -1863.379} C_VEL
LIN {X 0,Y 580.312,Z 265.218,A -85,B 0,C 180,E1 -1866.065,E2 -1866.065} C_VEL
LIN {X 0,Y 580.262,Z 273.467,A -85,B 0,C 180,E1 -1868.846,E2 -1868.846} C_VEL
LIN {X 0,Y 580.199,Z 281.919,A -85,B 0,C 180,E1 -1871.643,E2 -1871.643} C_VEL
LIN {X 0,Y 580.174,Z 290.823,A -85,B 0,C 180,E1 -1874.544,E2 -1874.544} C_VEL
LIN {X 0,Y 580.13,Z 299.728,A -85,B 0,C 180,E1 -1877.405,E2 -1877.405} C_VEL
LIN {X 0,Y 580.105,Z 300.493,A -85,B 0,C 180,E1 -1877.649,E2 -1877.649} C_VEL
LIN {X 0,Y 580.806,Z 306.387,A -85,B 0,C 180,E1 -1877.775,E2 -1877.775} C_VEL
LIN {X 0,Y 580.731,Z 318.509,A -85,B 0,C 180,E1 -1878.084,E2 -1878.084} C_VEL
LIN {X 0,Y 580.616,Z 330.325,A -85,B 0,C 180,E1 -1878.515,E2 -1878.515} C_VEL
LIN {X 0,Y 580.505,Z 342.216,A -85,B 0,C 180,E1 -1879.096,E2 -1879.096} C_VEL
LIN {X 0,Y 580.446,Z 353.484,A -85,B 0,C 180,E1 -1879.801,E2 -1879.801} C_VEL
LIN {X 0,Y 580.352,Z 363.65,A -85,B 0,C 180,E1 -1880.591,E2 -1880.591} C_VEL
LIN {X 0,Y 580.279,Z 372.789,A -85,B 0,C 180,E1 -1881.468,E2 -1881.468} C_VEL
LIN {X 0,Y 580.199,Z 381.691,A -85,B 0,C 180,E1 -1882.518,E2 -1882.518} C_VEL
LIN {X 0,Y 580.12,Z 388.468,A -85,B 0,C 180,E1 -1883.505,E2 -1883.505} C_VEL
LIN {X 0,Y 580.139,Z 393.681,A -85,B 0,C 180,E1 -1884.439,E2 -1884.439} C_VEL
LIN {X 0,Y 580.108,Z 398.372,A -85,B 0,C 180,E1 -1885.484,E2 -1885.484} C_VEL
LIN {X 0,Y 580.123,Z 401.957,A -85,B 0,C 180,E1 -1886.527,E2 -1886.527} C_VEL
LIN {X 0,Y 580.043,Z 403.809,A -85,B 0,C 180,E1 -1887.222,E2 -1887.222} C_VEL
LIN {X 0,Y 580.04,Z 405.199,A -85,B 0,C 180,E1 -1887.917,E2 -1887.917} C_VEL
LIN {X 0,Y 580.04,Z 406.785,A -85,B 0,C 180,E1 -1889.306,E2 -1889.306} C_VEL
LIN {X 0,Y 580.037,Z 407,A -85,B 0,C 180,E1 -1890,E2 -1890} C_VEL
LIN {X 0,Y 580.047,Z 406.186,A -85,B 0,C 180,E1 -1891.389,E2 -1891.389} C_VEL
LIN {X 0,Y 580.04,Z 405.2,A -85,B 0,C 180,E1 -1892.083,E2 -1892.083} C_VEL
LIN {X 0,Y 580.043,Z 403.81,A -85,B 0,C 180,E1 -1892.778,E2 -1892.778} C_VEL
LIN {X 0,Y 580.11,Z 400.896,A -85,B 0,C 180,E1 -1893.821,E2 -1893.821} C_VEL
LIN {X 0,Y 580.053,Z 396.949,A -85,B 0,C 180,E1 -1894.865,E2 -1894.865} C_VEL
LIN {X 0,Y 580.139,Z 390.878,A -85,B 0,C 180,E1 -1896.085,E2 -1896.085} C_VEL
LIN {X 0,Y 580.184,Z 384.238,A -85,B 0,C 180,E1 -1897.132,E2 -1897.132} C_VEL
LIN {X 0,Y 580.25,Z 375.992,A -85,B 0,C 180,E1 -1898.182,E2 -1898.182} C_VEL
LIN {X 0,Y 580.308,Z 367.54,A -85,B 0,C 180,E1 -1899.058,E2 -1899.058} C_VEL
LIN {X 0,Y 580.412,Z 357.1,A -85,B 0,C 180,E1 -1899.936,E2 -1899.936} C_VEL
LIN {X 0,Y 580.454,Z 346.759,A -85,B 0,C 180,E1 -1900.64,E2 -1900.64} C_VEL
LIN {X 0,Y 580.563,Z 335.595,A -85,B 0,C 180,E1 -1901.247,E2 -1901.247} C_VEL
LIN {X 0,Y 580.63,Z 323.774,A -85,B 0,C 180,E1 -1901.741,E2 -1901.741} C_VEL
LIN {X 0,Y 580.778,Z 310.359,A -85,B 0,C 180,E1 -1902.137,E2 -1902.137} C_VEL
LIN {X 0,Y 580.678,Z 304.098,A -85,B 0,C 180,E1 -1902.272,E2 -1902.272} C_VEL
LIN {X 0,Y 580.105,Z 300.493,A -85,B 0,C 180,E1 -1902.351,E2 -1902.351} C_VEL
LIN {X 0,Y 580.156,Z 291.936,A -85,B 0,C 180,E1 -1905.096,E2 -1905.096} C_VEL
LIN {X 0,Y 580.207,Z 283.032,A -85,B 0,C 180,E1 -1907.991,E2 -1907.991} C_VEL
LIN {X 0,Y 580.239,Z 275.241,A -85,B 0,C 180,E1 -1910.564,E2 -1910.564} C_VEL
LIN {X 0,Y 580.268,Z 267.974,A -85,B 0,C 180,E1 -1913.002,E2 -1913.002} C_VEL
LIN {X 0,Y 580.327,Z 260.678,A -85,B 0,C 180,E1 -1915.462,E2 -1915.462} C_VEL
LIN {X 0,Y 580.345,Z 251.647,A -85,B 0,C 180,E1 -1918.577,E2 -1918.577} C_VEL
LIN {X 0,Y 580.433,Z 243.88,A -85,B 0,C 180,E1 -1921.375,E2 -1921.375} C_VEL
LIN {X 0,Y 580.508,Z 237.239,A -85,B 0,C 180,E1 -1923.841,E2 -1923.841} C_VEL
LIN {X 0,Y 580.426,Z 232.212,A -85,B 0,C 180,E1 -1925.78,E2 -1925.78} C_VEL
LIN {X 0,Y 580.256,Z 231.209,A -85,B 0,C 180,E1 -1926.233,E2 -1926.233} C_VEL
LIN {X 0,Y 580.278,Z 231.205,A -85,B 0,C 180,E1 -1929.182,E2 -1929.182} C_VEL
LIN {X 0,Y 580.232,Z 231.204,A -85,B 0,C 180,E1 -1931.772,E2 -1931.772} C_VEL
LIN {X 0,Y 580.234,Z 231.211,A -85,B 0,C 180,E1 -1934.628,E2 -1934.628} C_VEL
LIN {X 0,Y 580.245,Z 231.202,A -85,B 0,C 180,E1 -1937.631,E2 -1937.631} C_VEL
LIN {X 0,Y 580.261,Z 231.203,A -85,B 0,C 180,E1 -1940.064,E2 -1940.064} C_VEL
LIN {X 0,Y 580.258,Z 231.202,A -85,B 0,C 180,E1 -1943.069,E2 -1943.069} C_VEL
LIN {X 0,Y 580.29,Z 231.204,A -85,B 0,C 180,E1 -1946.143,E2 -1946.143} C_VEL
LIN {X 0,Y 580.259,Z 231.204,A -85,B 0,C 180,E1 -1948.613,E2 -1948.613} C_VEL
LIN {X 0,Y 580.276,Z 231.198,A -85,B 0,C 180,E1 -1951.022,E2 -1951.022} C_VEL
LIN {X 0,Y 580.256,Z 231.207,A -85,B 0,C 180,E1 -1954.149,E2 -1954.149} C_VEL
LIN {X 0,Y 580.264,Z 231.201,A -85,B 0,C 180,E1 -1956.441,E2 -1956.441} C_VEL
LIN {X 0,Y 580.263,Z 231.206,A -85,B 0,C 180,E1 -1959.436,E2 -1959.436} C_VEL
LIN {X 0,Y 580.256,Z 231.21,A -85,B 0,C 180,E1 -1961.644,E2 -1961.644} C_VEL
LIN {X 0,Y 580.27,Z 231.204,A -85,B 0,C 180,E1 -1963.825,E2 -1963.825} C_VEL
LIN {X 0,Y 580.314,Z 231.196,A -85,B 0,C 180,E1 -1965.982,E2 -1965.982} C_VEL
LIN {X 0,Y 580.295,Z 231.199,A -85,B 0,C 180,E1 -1968.826,E2 -1968.826} C_VEL
LIN {X 0,Y 580.324,Z 231.195,A -85,B 0,C 180,E1 -1971.643,E2 -1971.643} C_VEL
LIN {X 0,Y 580.31,Z 231.196,A -85,B 0,C 180,E1 -1974.439,E2 -1974.439} C_VEL
LIN {X 0,Y 580.339,Z 231.196,A -85,B 0,C 180,E1 -1977.223,E2 -1977.223} C_VEL
LIN {X 0,Y 580.336,Z 231.192,A -85,B 0,C 180,E1 -1979.999,E2 -1979.999} C_VEL
LIN {X 0,Y 580.338,Z 231.199,A -85,B 0,C 180,E1 -1982.776,E2 -1982.776} C_VEL
LIN {X 0,Y 580.319,Z 231.193,A -85,B 0,C 180,E1 -1985.559,E2 -1985.559} C_VEL
LIN {X 0,Y 580.326,Z 231.201,A -85,B 0,C 180,E1 -1988.355,E2 -1988.355} C_VEL
LIN {X 0,Y 580.322,Z 231.193,A -85,B 0,C 180,E1 -1991.208,E2 -1991.208} C_VEL
LIN {X 0,Y 580.303,Z 231.202,A -85,B 0,C 180,E1 -1994.338,E2 -1994.338} C_VEL
LIN {X 0,Y 580.302,Z 231.195,A -85,B 0,C 180,E1 -1996.914,E2 -1996.914} C_VEL
LIN {X 0,Y 580.297,Z 231.204,A -85,B 0,C 180,E1 -1999.822,E2 -1999.822} C_VEL
LIN {X 0,Y 580.275,Z 231.2,A -85,B 0,C 180,E1 -2001.345,E2 -2001.345} C_VEL
LIN {X 0,Y 579.578,Z 231.294,A -85,B 0,C 180,E1 -2001.925,E2 -2001.925} C_VEL
LIN {X 0,Y 576.7,Z 231.648,A -85,B 0,C 180,E1 -2002.864,E2 -2002.864} C_VEL
LIN {X 0,Y 574.305,Z 231.949,A -85,B 0,C 180,E1 -2003.621,E2 -2003.621} C_VEL
LIN {X 0,Y 573.307,Z 232.07,A -85,B 0,C 180,E1 -2004.204,E2 -2004.204} C_VEL
LIN {X 0,Y 573.24,Z 232.076,A -85,B 0,C 180,E1 -2004.402,E2 -2004.402} C_VEL
LIN {X 0,Y 573.256,Z 232.074,A -85,B 0,C 180,E1 -2006.974,E2 -2006.974} C_VEL
LIN {X 0,Y 573.243,Z 232.084,A -85,B 0,C 180,E1 -2009.49,E2 -2009.49} C_VEL
LIN {X 0,Y 573.244,Z 232.075,A -85,B 0,C 180,E1 -2012.229,E2 -2012.229} C_VEL
LIN {X 0,Y 573.24,Z 232.077,A -85,B 0,C 180,E1 -2014.774,E2 -2014.774} C_VEL
LIN {X 0,Y 573.242,Z 232.084,A -85,B 0,C 180,E1 -2017.166,E2 -2017.166} C_VEL
LIN {X 0,Y 573.237,Z 232.077,A -85,B 0,C 180,E1 -2019.606,E2 -2019.606} C_VEL
LIN {X 0,Y 573.247,Z 232.078,A -85,B 0,C 180,E1 -2022.644,E2 -2022.644} C_VEL
LIN {X 0,Y 573.226,Z 232.076,A -85,B 0,C 180,E1 -2025.667,E2 -2025.667} C_VEL
LIN {X 0,Y 573.232,Z 232.083,A -85,B 0,C 180,E1 -2028.544,E2 -2028.544} C_VEL
LIN {X 0,Y 573.235,Z 232.076,A -85,B 0,C 180,E1 -2031.299,E2 -2031.299} C_VEL
LIN {X 0,Y 573.231,Z 232.079,A -85,B 0,C 180,E1 -2034.014,E2 -2034.014} C_VEL
LIN {X 0,Y 573.272,Z 232.078,A -85,B 0,C 180,E1 -2036.519,E2 -2036.519} C_VEL
LIN {X 0,Y 573.219,Z 232.078,A -85,B 0,C 180,E1 -2039.117,E2 -2039.117} C_VEL
LIN {X 0,Y 573.239,Z 232.082,A -85,B 0,C 180,E1 -2041.971,E2 -2041.971} C_VEL
LIN {X 0,Y 573.232,Z 232.078,A -85,B 0,C 180,E1 -2044.589,E2 -2044.589} C_VEL
LIN {X 0,Y 573.222,Z 232.077,A -85,B 0,C 180,E1 -2046.901,E2 -2046.901} C_VEL
LIN {X 0,Y 573.167,Z 232.09,A -85,B 0,C 180,E1 -2047.66,E2 -2047.66} C_VEL
LIN {X 0,Y 573.167,Z 234.317,A -85,B 0,C 180,E1 -2049.171,E2 -2049.171} C_VEL
LIN {X 0,Y 573.165,Z 238.064,A -85,B 0,C 180,E1 -2051.41,E2 -2051.41} C_VEL
LIN {X 0,Y 573.153,Z 241.801,A -85,B 0,C 180,E1 -2053.619,E2 -2053.619} C_VEL
LIN {X 0,Y 573.107,Z 246.781,A -85,B 0,C 180,E1 -2056.527,E2 -2056.527} C_VEL
LIN {X 0,Y 573.073,Z 251.795,A -85,B 0,C 180,E1 -2059.4,E2 -2059.4} C_VEL
LIN {X 0,Y 573.062,Z 256.867,A -85,B 0,C 180,E1 -2062.247,E2 -2062.247} C_VEL
LIN {X 0,Y 573.025,Z 260.8,A -85,B 0,C 180,E1 -2064.369,E2 -2064.369} C_VEL
LIN {X 0,Y 572.972,Z 266.098,A -85,B 0,C 180,E1 -2067.188,E2 -2067.188} C_VEL
LIN {X 0,Y 572.977,Z 271.455,A -85,B 0,C 180,E1 -2070,E2 -2070} C_VEL
LIN {X 0,Y 572.977,Z 272.551,A -85,B 0,C 180,E1 -2070.571,E2 -2070.571} C_VEL
LIN {X 0,Y 573.84,Z 278.919,A -85,B 0,C 180,E1 -2070.724,E2 -2070.724} C_VEL
LIN {X 0,Y 573.722,Z 291.937,A -85,B 0,C 180,E1 -2071.097,E2 -2071.097} C_VEL
LIN {X 0,Y 573.574,Z 303.92,A -85,B 0,C 180,E1 -2071.58,E2 -2071.58} C_VEL
LIN {X 0,Y 573.498,Z 315.487,A -85,B 0,C 180,E1 -2072.195,E2 -2072.195} C_VEL
LIN {X 0,Y 573.405,Z 327.091,A -85,B 0,C 180,E1 -2072.986,E2 -2072.986} C_VEL
LIN {X 0,Y 573.285,Z 337.445,A -85,B 0,C 180,E1 -2073.866,E2 -2073.866} C_VEL
LIN {X 0,Y 573.177,Z 345.873,A -85,B 0,C 180,E1 -2074.747,E2 -2074.747} C_VEL
LIN {X 0,Y 573.11,Z 354.114,A -85,B 0,C 180,E1 -2075.806,E2 -2075.806} C_VEL
LIN {X 0,Y 573.04,Z 361.778,A -85,B 0,C 180,E1 -2077.045,E2 -2077.045} C_VEL
LIN {X 0,Y 573.03,Z 366.9,A -85,B 0,C 180,E1 -2078.108,E2 -2078.108} C_VEL
LIN {X 0,Y 572.968,Z 370.891,A -85,B 0,C 180,E1 -2079.175,E2 -2079.175} C_VEL
LIN {X 0,Y 572.977,Z 372.944,A -85,B 0,C 180,E1 -2079.888,E2 -2079.888} C_VEL
LIN {X 0,Y 573.023,Z 375.522,A -85,B 0,C 180,E1 -2081.14,E2 -2081.14} C_VEL
LIN {X 0,Y 572.939,Z 376.579,A -85,B 0,C 180,E1 -2082.036,E2 -2082.036} C_VEL
LIN {X 0,Y 572.94,Z 376.942,A -85,B 0,C 180,E1 -2082.756,E2 -2082.756} C_VEL
LIN {X 0,Y 572.961,Z 376.91,A -85,B 0,C 180,E1 -2083.477,E2 -2083.477} C_VEL
LIN {X 0,Y 572.965,Z 376.346,A -85,B 0,C 180,E1 -2084.306,E2 -2084.306} C_VEL
LIN {X 0,Y 572.951,Z 374.233,A -85,B 0,C 180,E1 -2085.655,E2 -2085.655} C_VEL
LIN {X 0,Y 572.998,Z 370.848,A -85,B 0,C 180,E1 -2086.928,E2 -2086.928} C_VEL
LIN {X 0,Y 572.995,Z 367.411,A -85,B 0,C 180,E1 -2087.856,E2 -2087.856} C_VEL
LIN {X 0,Y 573.068,Z 362.474,A -85,B 0,C 180,E1 -2088.911,E2 -2088.911} C_VEL
LIN {X 0,Y 573.087,Z 355.517,A -85,B 0,C 180,E1 -2090.082,E2 -2090.082} C_VEL
LIN {X 0,Y 573.147,Z 348.268,A -85,B 0,C 180,E1 -2091.057,E2 -2091.057} C_VEL
LIN {X 0,Y 573.252,Z 340.142,A -85,B 0,C 180,E1 -2091.957,E2 -2091.957} C_VEL
LIN {X 0,Y 573.366,Z 329.686,A -85,B 0,C 180,E1 -2092.902,E2 -2092.902} C_VEL
LIN {X 0,Y 573.435,Z 319.17,A -85,B 0,C 180,E1 -2093.665,E2 -2093.665} C_VEL
LIN {X 0,Y 573.578,Z 307.585,A -85,B 0,C 180,E1 -2094.33,E2 -2094.33} C_VEL
LIN {X 0,Y 573.699,Z 296.504,A -85,B 0,C 180,E1 -2094.825,E2 -2094.825} C_VEL
LIN {X 0,Y 573.854,Z 283.19,A -85,B 0,C 180,E1 -2095.261,E2 -2095.261} C_VEL
LIN {X 0,Y 573.706,Z 277.094,A -85,B 0,C 180,E1 -2095.41,E2 -2095.41} C_VEL
LIN {X 0,Y 572.971,Z 272.549,A -85,B 0,C 180,E1 -2095.52,E2 -2095.52} C_VEL
LIN {X 0,Y 572.968,Z 266.712,A -85,B 0,C 180,E1 -2098.578,E2 -2098.578} C_VEL
LIN {X 0,Y 572.966,Z 262.134,A -85,B 0,C 180,E1 -2101.008,E2 -2101.008} C_VEL
LIN {X 0,Y 573.015,Z 257.505,A -85,B 0,C 180,E1 -2103.498,E2 -2103.498} C_VEL
LIN {X 0,Y 573.049,Z 252.91,A -85,B 0,C 180,E1 -2106.063,E2 -2106.063} C_VEL
LIN {X 0,Y 573.072,Z 248.307,A -85,B 0,C 180,E1 -2108.714,E2 -2108.714} C_VEL
LIN {X 0,Y 573.091,Z 243.369,A -85,B 0,C 180,E1 -2111.579,E2 -2111.579} C_VEL
LIN {X 0,Y 573.178,Z 238.117,A -85,B 0,C 180,E1 -2114.672,E2 -2114.672} C_VEL
LIN {X 0,Y 573.201,Z 233.261,A -85,B 0,C 180,E1 -2117.598,E2 -2117.598} C_VEL
LIN {X 0,Y 573.193,Z 232.088,A -85,B 0,C 180,E1 -2118.541,E2 -2118.541} C_VEL
LIN {X 0,Y 573.229,Z 232.082,A -85,B 0,C 180,E1 -2120.569,E2 -2120.569} C_VEL
LIN {X 0,Y 573.244,Z 232.08,A -85,B 0,C 180,E1 -2123.078,E2 -2123.078} C_VEL
LIN {X 0,Y 573.256,Z 232.082,A -85,B 0,C 180,E1 -2125.672,E2 -2125.672} C_VEL
LIN {X 0,Y 573.236,Z 232.08,A -85,B 0,C 180,E1 -2128.186,E2 -2128.186} C_VEL
LIN {X 0,Y 573.261,Z 232.078,A -85,B 0,C 180,E1 -2130.635,E2 -2130.635} C_VEL
LIN {X 0,Y 573.234,Z 232.081,A -85,B 0,C 180,E1 -2133.024,E2 -2133.024} C_VEL
LIN {X 0,Y 573.261,Z 232.076,A -85,B 0,C 180,E1 -2135.367,E2 -2135.367} C_VEL
LIN {X 0,Y 573.246,Z 232.081,A -85,B 0,C 180,E1 -2137.664,E2 -2137.664} C_VEL
LIN {X 0,Y 573.254,Z 232.08,A -85,B 0,C 180,E1 -2140.671,E2 -2140.671} C_VEL
LIN {X 0,Y 573.249,Z 232.08,A -85,B 0,C 180,E1 -2143.623,E2 -2143.623} C_VEL
LIN {X 0,Y 573.214,Z 232.083,A -85,B 0,C 180,E1 -2146.53,E2 -2146.53} C_VEL
LIN {X 0,Y 573.249,Z 232.079,A -85,B 0,C 180,E1 -2148.746,E2 -2148.746} C_VEL
LIN {X 0,Y 573.297,Z 232.076,A -85,B 0,C 180,E1 -2151.542,E2 -2151.542} C_VEL
LIN {X 0,Y 573.276,Z 232.079,A -85,B 0,C 180,E1 -2154.373,E2 -2154.373} C_VEL
LIN {X 0,Y 573.307,Z 232.073,A -85,B 0,C 180,E1 -2157.19,E2 -2157.19} C_VEL
LIN {X 0,Y 573.299,Z 232.072,A -85,B 0,C 180,E1 -2160.001,E2 -2160.001} C_VEL
LIN {X 0,Y 573.302,Z 232.071,A -85,B 0,C 180,E1 -2162.811,E2 -2162.811} C_VEL
LIN {X 0,Y 573.278,Z 232.074,A -85,B 0,C 180,E1 -2165.629,E2 -2165.629} C_VEL
LIN {X 0,Y 573.275,Z 232.075,A -85,B 0,C 180,E1 -2168.46,E2 -2168.46} C_VEL
LIN {X 0,Y 573.29,Z 232.075,A -85,B 0,C 180,E1 -2171.312,E2 -2171.312} C_VEL
LIN {X 0,Y 573.257,Z 232.078,A -85,B 0,C 180,E1 -2174.42,E2 -2174.42} C_VEL
LIN {X 0,Y 573.252,Z 232.083,A -85,B 0,C 180,E1 -2177.113,E2 -2177.113} C_VEL
LIN {X 0,Y 573.231,Z 232.086,A -85,B 0,C 180,E1 -2180.078,E2 -2180.078} C_VEL
LIN {X 0,Y 573.227,Z 232.081,A -85,B 0,C 180,E1 -2182.339,E2 -2182.339} C_VEL
LIN {X 0,Y 573.249,Z 232.078,A -85,B 0,C 180,E1 -2185.411,E2 -2185.411} C_VEL
LIN {X 0,Y 573.218,Z 232.082,A -85,B 0,C 180,E1 -2188.566,E2 -2188.566} C_VEL
LIN {X 0,Y 573.231,Z 232.082,A -85,B 0,C 180,E1 -2190.994,E2 -2190.994} C_VEL
LIN {X 0,Y 573.257,Z 232.08,A -85,B 0,C 180,E1 -2193.525,E2 -2193.525} C_VEL
LIN {X 0,Y 573.209,Z 232.082,A -85,B 0,C 180,E1 -2196.053,E2 -2196.053} C_VEL
LIN {X 0,Y 573.244,Z 232.079,A -85,B 0,C 180,E1 -2198.702,E2 -2198.702} C_VEL
LIN {X 0,Y 573.222,Z 232.082,A -85,B 0,C 180,E1 -2201.593,E2 -2201.593} C_VEL
LIN {X 0,Y 573.236,Z 232.082,A -85,B 0,C 180,E1 -2204.334,E2 -2204.334} C_VEL
LIN {X 0,Y 573.217,Z 232.087,A -85,B 0,C 180,E1 -2207.362,E2 -2207.362} C_VEL
LIN {X 0,Y 573.247,Z 232.083,A -85,B 0,C 180,E1 -2210.394,E2 -2210.394} C_VEL
LIN {X 0,Y 573.251,Z 232.082,A -85,B 0,C 180,E1 -2213.079,E2 -2213.079} C_VEL
LIN {X 0,Y 573.237,Z 232.21,A -85,B 0,C 180,E1 -2213.679,E2 -2213.679} C_VEL
LIN {X 0,Y 573.532,Z 235.929,A -85,B 0,C 180,E1 -2215.187,E2 -2215.187} C_VEL
LIN {X 0,Y 573.484,Z 242.566,A -85,B 0,C 180,E1 -2217.736,E2 -2217.736} C_VEL
LIN {X 0,Y 573.382,Z 250.486,A -85,B 0,C 180,E1 -2220.642,E2 -2220.642} C_VEL
LIN {X 0,Y 573.277,Z 258.546,A -85,B 0,C 180,E1 -2223.5,E2 -2223.5} C_VEL
LIN {X 0,Y 573.262,Z 266.249,A -85,B 0,C 180,E1 -2226.137,E2 -2226.137} C_VEL
LIN {X 0,Y 573.235,Z 273.883,A -85,B 0,C 180,E1 -2228.715,E2 -2228.715} C_VEL
LIN {X 0,Y 573.159,Z 281.919,A -85,B 0,C 180,E1 -2231.41,E2 -2231.41} C_VEL
LIN {X 0,Y 573.107,Z 290.823,A -85,B 0,C 180,E1 -2234.349,E2 -2234.349} C_VEL
LIN {X 0,Y 573.065,Z 299.728,A -85,B 0,C 180,E1 -2237.247,E2 -2237.247} C_VEL
LIN {X 0,Y 573.045,Z 300.493,A -85,B 0,C 180,E1 -2237.494,E2 -2237.494} C_VEL
LIN {X 0,Y 573.874,Z 306.386,A -85,B 0,C 180,E1 -2237.625,E2 -2237.625} C_VEL
LIN {X 0,Y 573.771,Z 318.51,A -85,B 0,C 180,E1 -2237.937,E2 -2237.937} C_VEL
LIN {X 0,Y 573.65,Z 330.323,A -85,B 0,C 180,E1 -2238.374,E2 -2238.374} C_VEL
LIN {X 0,Y 573.511,Z 342.653,A -85,B 0,C 180,E1 -2238.986,E2 -2238.986} C_VEL
LIN {X 0,Y 573.442,Z 353.486,A -85,B 0,C 180,E1 -2239.675,E2 -2239.675} C_VEL
LIN {X 0,Y 573.307,Z 363.65,A -85,B 0,C 180,E1 -2240.474,E2 -2240.474} C_VEL
LIN {X 0,Y 573.215,Z 372.789,A -85,B 0,C 180,E1 -2241.362,E2 -2241.362} C_VEL
LIN {X 0,Y 573.143,Z 381.691,A -85,B 0,C 180,E1 -2242.426,E2 -2242.426} C_VEL
LIN {X 0,Y 573.051,Z 388.407,A -85,B 0,C 180,E1 -2243.415,E2 -2243.415} C_VEL
LIN {X 0,Y 573.07,Z 393.681,A -85,B 0,C 180,E1 -2244.37,E2 -2244.37} C_VEL
LIN {X 0,Y 573.028,Z 398.373,A -85,B 0,C 180,E1 -2245.428,E2 -2245.428} C_VEL
LIN {X 0,Y 573.022,Z 401.958,A -85,B 0,C 180,E1 -2246.484,E2 -2246.484} C_VEL
LIN {X 0,Y 572.959,Z 403.808,A -85,B 0,C 180,E1 -2247.188,E2 -2247.188} C_VEL
LIN {X 0,Y 572.94,Z 405.198,A -85,B 0,C 180,E1 -2247.891,E2 -2247.891} C_VEL
LIN {X 0,Y 572.941,Z 406.785,A -85,B 0,C 180,E1 -2249.297,E2 -2249.297} C_VEL
LIN {X 0,Y 572.938,Z 407,A -85,B 0,C 180,E1 -2250,E2 -2250} C_VEL
LIN {X 0,Y 572.946,Z 406.186,A -85,B 0,C 180,E1 -2251.406,E2 -2251.406} C_VEL
LIN {X 0,Y 572.94,Z 405.199,A -85,B 0,C 180,E1 -2252.109,E2 -2252.109} C_VEL
LIN {X 0,Y 572.959,Z 403.81,A -85,B 0,C 180,E1 -2252.812,E2 -2252.812} C_VEL
LIN {X 0,Y 573.015,Z 400.896,A -85,B 0,C 180,E1 -2253.868,E2 -2253.868} C_VEL
LIN {X 0,Y 572.963,Z 396.949,A -85,B 0,C 180,E1 -2254.926,E2 -2254.926} C_VEL
LIN {X 0,Y 573.065,Z 390.877,A -85,B 0,C 180,E1 -2256.16,E2 -2256.16} C_VEL
LIN {X 0,Y 573.12,Z 384.238,A -85,B 0,C 180,E1 -2257.221,E2 -2257.221} C_VEL
LIN {X 0,Y 573.201,Z 375.992,A -85,B 0,C 180,E1 -2258.283,E2 -2258.283} C_VEL
LIN {X 0,Y 573.287,Z 367.54,A -85,B 0,C 180,E1 -2259.17,E2 -2259.17} C_VEL
LIN {X 0,Y 573.405,Z 357.101,A -85,B 0,C 180,E1 -2260.058,E2 -2260.058} C_VEL
LIN {X 0,Y 573.519,Z 345.539,A -85,B 0,C 180,E1 -2260.847,E2 -2260.847} C_VEL
LIN {X 0,Y 573.609,Z 333.889,A -85,B 0,C 180,E1 -2261.466,E2 -2261.466} C_VEL
LIN {X 0,Y 573.763,Z 321.179,A -85,B 0,C 180,E1 -2261.974,E2 -2261.974} C_VEL
LIN {X 0,Y 573.854,Z 308.529,A -85,B 0,C 180,E1 -2262.331,E2 -2262.331} C_VEL
LIN {X 0,Y 573.675,Z 304.661,A -85,B 0,C 180,E1 -2262.413,E2 -2262.413} C_VEL
LIN {X 0,Y 573.045,Z 300.493,A -85,B 0,C 180,E1 -2262.506,E2 -2262.506} C_VEL
LIN {X 0,Y 573.085,Z 291.936,A -85,B 0,C 180,E1 -2265.287,E2 -2265.287} C_VEL
LIN {X 0,Y 573.146,Z 284.145,A -85,B 0,C 180,E1 -2267.851,E2 -2267.851} C_VEL
LIN {X 0,Y 573.196,Z 276.354,A -85,B 0,C 180,E1 -2270.453,E2 -2270.453} C_VEL
LIN {X 0,Y 573.216,Z 268.392,A -85,B 0,C 180,E1 -2273.139,E2 -2273.139} C_VEL
LIN {X 0,Y 573.28,Z 260.584,A -85,B 0,C 180,E1 -2275.798,E2 -2275.798} C_VEL
LIN {X 0,Y 573.327,Z 252.716,A -85,B 0,C 180,E1 -2278.559,E2 -2278.559} C_VEL
LIN {X 0,Y 573.425,Z 244.941,A -85,B 0,C 180,E1 -2281.391,E2 -2281.391} C_VEL
LIN {X 0,Y 573.527,Z 239.156,A -85,B 0,C 180,E1 -2283.563,E2 -2283.563} C_VEL
LIN {X 0,Y 573.523,Z 233.959,A -85,B 0,C 180,E1 -2285.575,E2 -2285.575} C_VEL
LIN {X 0,Y 573.232,Z 232.084,A -85,B 0,C 180,E1 -2286.376,E2 -2286.376} C_VEL
LIN {X 0,Y 573.229,Z 232.08,A -85,B 0,C 180,E1 -2289.429,E2 -2289.429} C_VEL
LIN {X 0,Y 573.188,Z 232.083,A -85,B 0,C 180,E1 -2291.587,E2 -2291.587} C_VEL
LIN {X 0,Y 573.208,Z 232.082,A -85,B 0,C 180,E1 -2294.335,E2 -2294.335} C_VEL
LIN {X 0,Y 573.204,Z 232.08,A -85,B 0,C 180,E1 -2297.361,E2 -2297.361} C_VEL
LIN {X 0,Y 573.221,Z 232.085,A -85,B 0,C 180,E1 -2300.39,E2 -2300.39} C_VEL
LIN {X 0,Y 573.213,Z 232.079,A -85,B 0,C 180,E1 -2303.074,E2 -2303.074} C_VEL
LIN {X 0,Y 573.248,Z 232.075,A -85,B 0,C 180,E1 -2305.669,E2 -2305.669} C_VEL
LIN {X 0,Y 573.228,Z 232.085,A -85,B 0,C 180,E1 -2308.183,E2 -2308.183} C_VEL
